// TwinCAT 3 PLC project PLC1
// ProgramVersion: 3.1.4026.19
// libraries:
//   Tc2_ControllerToolbox, * (Beckhoff Automation GmbH)
//   Tc2_PfwLib_Processing, * (Beckhoff Automation GmbH)
//   Tc2_Standard, * (Beckhoff Automation GmbH)
//   Tc2_System, * (Beckhoff Automation GmbH)
//   Tc2_Utilities, * (Beckhoff Automation GmbH)
//   Tc3_Module, * (Beckhoff Automation GmbH)
//   VisuDialogs, * (System)
// project tree:
//   / MAIN.TcPOU, MAIN_Fast.TcPOU, Visualization Manager.TcVMO (not stored)
//   Tasks/ Fast_Task.TcTTO, PLC_Task.TcTTO (not stored), Temperature_Task.TcTTO (not stored)
//   Temperature/DUTs/ E_HMIstatus.TcDUT, E_MainStateMachine.TcDUT, ST_TempLoad.TcDUT, ST_TempLoad_Cmd.TcDUT, ST_TempLoad_State.TcDUT, ST_TempSave.TcDUT, ST_TempSave_Cmd.TcDUT (not stored)
//   Temperature/ FB_Load.TcPOU, FB_MainVisu.TcPOU, FB_Save.TcPOU, TemperatureCtrl.TcPOU
//   Temperature/GVLs/ GVL_10_Visu.TcGVL (not stored), GVL_20_Application.TcGVL, GVL_30_Scope.TcGVL (not stored)
//   Temperature/TextLists/ GlobalTextList_1.TcGTLO (not stored), TL_Mparams_LREAL.TcTLO, TL_Params_BOOL.TcTLO (not stored), TL_Params_Enum.TcTLO (not stored), TL_Params_INT.TcTLO, TL_Pparmas.TcTLO (not stored), TL_Supply.TcTLO, TL_TcPfw_ErrorId.TcTLO, TL_TctrlOutSelect.TcTLO (not stored), TL_TctrlPowerTerminal.TcTLO (not stored), TL_TempSensType.TcTLO, TL_TerminalType.TcTLO (not stored)
//   Temperature/VISUs/DUTs/ st_ParamsUnsave.TcDUT (not stored), ST_Param_Visu.TcDUT (not stored)
//   Temperature/VISUs/POUs/ FB_Visu_Param.TcPOU (not stored), FB_Visu_Pparam.TcPOU (not stored), FB_Visu_Supply.TcPOU (not stored)
//   Temperature/VISUs/VISUs/Pages/Load Save/ Visu_SaveLoad.TcVIS
//   Temperature/VISUs/VISUs/Pages/LoopTest/ Visu_LoopTest.TcVIS
//   Temperature/VISUs/VISUs/Pages/Machine/Parameter/ Param_BOOL.TcVIS, Param_DINT.TcVIS, Param_ENUM_PowerTerm.TcVIS, Param_ENUM_SelOut.TcVIS, Param_ENUM_SensType.TcVIS, Param_ENUM_TermType.TcVIS, Param_LREAL.TcVIS
//   Temperature/VISUs/VISUs/Pages/Machine/Subpage/ Visu_Mparam_Autotune.TcVIS, Visu_Mparam_Cool.TcVIS, Visu_Mparam_Extruder.TcVIS (excluded from build), Visu_Mparam_General.TcVIS, Visu_Mparam_Heat.TcVIS, Visu_Mparam_Supply.TcVIS, Visu_Mparam_Temperature.TcVIS
//   Temperature/VISUs/VISUs/Pages/Machine/ Visu_MParam.TcVIS
//   Temperature/VISUs/VISUs/Pages/Product/ Param_LREAL_Pparam.TcVIS, Visu_PParam.TcVIS, Visu_PParam_Params.TcVIS
//   Temperature/VISUs/VISUs/Pages/Supply/ Param_LREAL_Supply.TcVIS, Visu_Supply.TcVIS, Visu_Supply_Params.TcVIS
//   Temperature/VISUs/VISUs/Pages/ Visu_Main.TcVIS
//   Utility/Linearisation/ FB_Linear_Interpolation.TcPOU
//   Utility/Ramp Generator/ FB_Ramp_Generator.TcPOU, ST_Ramp_Generator.TcDUT
//   Utility/Setpoint Generator/ FB_Setpoint_Generator.TcPOU, ST_Setpoint_Generator.TcDUT
// real-time tasks:
//   TASK Temperature Task: cycle T#25000us, priority 20, ADS port 350
//   TASK PLC Task: cycle T#10ms, priority 1, ADS port 351
//   TASK Fast Task: cycle T#2ms, priority 2, ADS port 352
// I/O:
//   DEVICE Device 1 (EtherCAT) (disabled), AmsNetId 5.70.226.154.2.1
//     Term 1 (EK1200) [EK1200-5000 EtherCAT Power supply (2A E-Bus)]
//       Term 2 (EL3202) [EL3202 2Ch. Ana. Input PT100 (RTD)]
//       Term 3 (EL1809) [EL1809 16Ch. Dig. Input 24V, 3ms]
//       Term 4 (EL2809) [EL2809 16Ch. Dig. Output 24V, 0.5A]
//       Term 5 (EL9011) [EL9011 End Terminal]
//   DEVICE Device 2 (EtherCAT Automation Protocol) (disabled), AmsNetId 5.77.2.52.3.1
//     Box 6 (Publisher)
//     Box 7 (Subscriber)

CONFIGURATION PLC1
    RESOURCE PLC ON TwinCAT3
        TASK Fast_Task(INTERVAL := T#2ms, PRIORITY := 2);
        PROGRAM MAIN_Fast WITH Fast_Task : MAIN_Fast;
    END_RESOURCE
END_CONFIGURATION

// ---- Temperature/DUTs/E_HMIstatus.TcDUT
TYPE E_HMIstatus :
(
	Off 				:= 0,
	Standby,
	On,
	Autotune,
	IdleLoad
);
END_TYPE

// ---- Temperature/DUTs/E_MainStateMachine.TcDUT
TYPE E_MainStateMachine :
(
	eMainSM_BasicInit 						:= 0,
	eMainSM_TempInit,
	eMainSM_MParamLoad,
	eMainSM_PParamLoad,
	eMainSM_SupParamLoad,
	eMainSM_StartUp,
	eMainSM_Idle
);
END_TYPE

// ---- Temperature/DUTs/ST_TempLoad.TcDUT
TYPE ST_TempLoad :
STRUCT
	stTempCmd						: ST_TempLoad_Cmd;
	stTempState						: ST_TempLoad_State;
END_STRUCT
END_TYPE

// ---- Temperature/DUTs/ST_TempLoad_Cmd.TcDUT
TYPE ST_TempLoad_Cmd :
STRUCT
	bLoadPparams							: BOOL;
	bLoadMparams							: BOOL;
	bLoadSupplyParams						: BOOL;
END_STRUCT
END_TYPE

// ---- Temperature/DUTs/ST_TempLoad_State.TcDUT
TYPE ST_TempLoad_State :
STRUCT
	bPparamLoaded									: BOOL;
	bMparamLoaded									: BOOL;
	bPparamLoad										: BOOL;
	bMparamLoad										: BOOL;
	bSupplyParamsLoad								: BOOL;
	bSupplyParamsLoaded								: BOOL;
END_STRUCT
END_TYPE

// ---- Temperature/DUTs/ST_TempSave.TcDUT
TYPE ST_TempSave :
STRUCT
	stTempCmd							: ST_TempSave_Cmd;
END_STRUCT
END_TYPE

// ---- Utility/Ramp Generator/ST_Ramp_Generator.TcDUT
TYPE ST_Ramp_Generator :
STRUCT
	tRefreshRate									: LREAL;
	fVelPos											: LREAL	:= 20;
	fVelNeg											: LREAL	:= 40;
END_STRUCT
END_TYPE

// ---- Utility/Setpoint Generator/ST_Setpoint_Generator.TcDUT
TYPE ST_Setpoint_Generator :
STRUCT
	tRefreshRate									: LREAL;
	bDisableRamping									: BOOL	:= FALSE;(*A continuous output value is not calculated if this parameter is TRUE. There is a step change between the output values*)
END_STRUCT
END_TYPE

// ---- Temperature/GVLs/GVL_20_Application.TcGVL
VAR_GLOBAL
	stTempLoad				: ST_TempLoad;
	stTempSave				: ST_TempSave;
END_VAR

// ---- MAIN_Fast.TcPOU
PROGRAM MAIN_Fast
VAR
	fbGetCurTaskIdx 			: GETCURTASKINDEX;
	bFirstCycle					: BOOL;
//	For temperature feedback linearisation
	fbLinInterpolation			: FB_Linear_Interpolation;
//	Setpoint generator
	fbSetpointGenerator			: FB_Setpoint_Generator;
//	Ramp generator
	fbRampGenerator				: FB_Ramp_Generator;
END_VAR


// =========================================================
	// Get plc task first cycle flag	
fbGetCurTaskIdx(); 
bFirstCycle:= _TaskInfo[fbGetCurTaskIdx.index].FirstCycle;

IF bFirstCycle THEN
	;
END_IF

	// Temperature feedback linearisation	
fbLinInterpolation();	
fbLinInterpolation.M_Cyclic();

	// Setpoint generator	
fbSetpointGenerator();
fbSetpointGenerator.M_Cyclic();	
	// Ramp generator
fbRampGenerator();
fbRampGenerator.M_Cyclic();
	
// =========================================================

END_PROGRAM

// ---- Utility/Linearisation/FB_Linear_Interpolation.TcPOU
FUNCTION_BLOCK FB_Linear_Interpolation
VAR CONSTANT
	nNoOfRows											: INT:= 45;
	nNoOfColumns										: INT:= 2;
END_VAR
VAR
	arrTableOffset										: ARRAY[1..nNoOfRows,1..nNoOfColumns] OF LREAL;	
	arrTable											: ARRAY[1..nNoOfRows,1..nNoOfColumns] OF LREAL;
	fIn, fOut, fManValue								: LREAL;
	bExtrapolate										: BOOL;
	eMode												: E_CTRL_MODE;
	stCTRL_LIN_INTERPOLATION_PARAMS						: ST_CTRL_LIN_INTERPOLATION_PARAMS;
	eErrorId											: E_CTRL_ERRORCODES;
	bError												: BOOL;
	fbCTRL_LIN_INTERPOLATION							: FB_CTRL_LIN_INTERPOLATION;
	bInit, bUpdate										: BOOL	:= TRUE;
	fbGetCurTaskIdx 									: GETCURTASKINDEX;
	bFirstCycle											: BOOL;
	fCycleTime											: LREAL := 0.025;
END_VAR

// =========================================================
	// Get temperature task first cycle flag	
fbGetCurTaskIdx(); 
bFirstCycle:= _TaskInfo[fbGetCurTaskIdx.index].FirstCycle;

IF bFirstCycle THEN
	;
END_IF

// Get Cycle Time
IF(GETCURTASKINDEXEX()<=0)THEN
	fCycletime:= TO_LREAL(0.025);(* Don't know, just guessing *)
ELSE
	fCycletime:= UDINT_TO_LREAL(_TaskInfo[GETCURTASKINDEXEX()].cycleTime)/10000000.0;
END_IF

// =========================================================

//FB_Init is always available implicitly and it is used primarily for initialization.
//The return value is not evaluated. For a specific influence, you can also declare the
//methods explicitly and provide additional code there with the standard initialization
//code. You can evaluate the return value.
METHOD FB_Init: BOOL
VAR_INPUT
    bInitRetains: BOOL; // TRUE: the retain variables are initialized (reset warm / reset cold)
    bInCopyCode: BOOL;  // TRUE: the instance will be copied to the copy code afterward (online change)   
END_VAR
// =========================================================
	// Init
	arrTableOffset[1,1]:= 0.1;		arrTableOffset[1,2]:= 0.9;
	arrTableOffset[2,1]:= 0.3;		arrTableOffset[2,2]:= 0.8;
	arrTableOffset[3,1]:= 0.5;		arrTableOffset[3,2]:= 0.7;
	arrTableOffset[4,1]:= 0.7;		arrTableOffset[4,2]:= 0.6;
	arrTableOffset[5,1]:= 0.9;		arrTableOffset[5,2]:= 0.5;
	arrTableOffset[6,1]:= 0.8;		arrTableOffset[6,2]:= 0.4;
	arrTableOffset[7,1]:= 0.7;		arrTableOffset[7,2]:= 0.3;
	arrTableOffset[8,1]:= 0.6;		arrTableOffset[8,2]:= 0.2;
	arrTableOffset[9,1]:= 0.5;		arrTableOffset[9,2]:= 0.1;
	arrTableOffset[10,1]:= 0.4;		arrTableOffset[10,2]:= 0.3;
	arrTableOffset[11,1]:= 0.3;		arrTableOffset[11,2]:= 0.5;
	arrTableOffset[12,1]:= 0.2;		arrTableOffset[12,2]:= 0.7;
	arrTableOffset[13,1]:= 0.1;		arrTableOffset[13,2]:= 0.9;
	arrTableOffset[14,1]:= 0.3;		arrTableOffset[14,2]:= 0.7;
	arrTableOffset[15,1]:= 0.5;		arrTableOffset[15,2]:= 0.5;
	arrTableOffset[16,1]:= 0.7;		arrTableOffset[16,2]:= 0.3;
	arrTableOffset[17,1]:= 0.9;		arrTableOffset[17,2]:= 0.1;
	arrTableOffset[18,1]:= 0.8;		arrTableOffset[18,2]:= 0.2;
	arrTableOffset[19,1]:= 0.7;		arrTableOffset[19,2]:= 0.3;
	arrTableOffset[20,1]:= 0.6;		arrTableOffset[20,2]:= 0.4;
	arrTableOffset[21,1]:= 0.5;		arrTableOffset[21,2]:= 0.5;
	arrTableOffset[22,1]:= 0.4;		arrTableOffset[22,2]:= 0.6;
	arrTableOffset[23,1]:= 0.3;		arrTableOffset[23,2]:= 0.7;
	arrTableOffset[24,1]:= 0.2;		arrTableOffset[24,2]:= 0.8;
	arrTableOffset[25,1]:= 0.1;		arrTableOffset[25,2]:= 0.9;
	arrTableOffset[26,1]:= 0.9;		arrTableOffset[26,2]:= 0.7;
	arrTableOffset[27,1]:= 0.7;		arrTableOffset[27,2]:= 0.5;
	arrTableOffset[28,1]:= 0.5;		arrTableOffset[28,2]:= 0.5;
	arrTableOffset[29,1]:= 0.3;		arrTableOffset[29,2]:= 0.3;
	arrTableOffset[30,1]:= 0.1;		arrTableOffset[30,2]:= 0.1;
	arrTableOffset[31,1]:= 0.3;		arrTableOffset[31,2]:= 0.3;
	arrTableOffset[32,1]:= 0.5;		arrTableOffset[32,2]:= 0.5;
	arrTableOffset[33,1]:= 0.7;		arrTableOffset[33,2]:= 0.7;
	arrTableOffset[34,1]:= 0.9;		arrTableOffset[34,2]:= 0.9;
	arrTableOffset[35,1]:= 0.8;		arrTableOffset[35,2]:= 0.7;
	arrTableOffset[36,1]:= 0.7;		arrTableOffset[36,2]:= 0.5;
	arrTableOffset[37,1]:= 0.6;		arrTableOffset[37,2]:= 0.3;
	arrTableOffset[38,1]:= 0.5;		arrTableOffset[38,2]:= 0.1;
	arrTableOffset[39,1]:= 0.4;		arrTableOffset[39,2]:= 0.2;
	arrTableOffset[40,1]:= 0.3;		arrTableOffset[40,2]:= 0.3;
	arrTableOffset[41,1]:= 0.2;		arrTableOffset[41,2]:= 0.4;
	arrTableOffset[42,1]:= 0.1;		arrTableOffset[42,2]:= 0.5;
	arrTableOffset[43,1]:= 0.3;		arrTableOffset[43,2]:= 0.6;
	arrTableOffset[44,1]:= 0.5;		arrTableOffset[44,2]:= 0.7;
	arrTableOffset[45,1]:= 0.7;		arrTableOffset[45,2]:= 0.8;
	
// =========================================================
END_METHOD

METHOD PUBLIC M_Cyclic
VAR_INPUT
END_VAR
// =========================================================
bUpdate := TRUE;

IF bInit OR bUpdate THEN
	(* Init array with the interpolation points  *)
	(* 	fIn					 						|		fOut		*)
	arrTable[1,1] := 25.0+arrTableOffset[1,1];			arrTable[1,2] := 25.0+arrTableOffset[1,2];
	arrTable[2,1] := 30.0+arrTableOffset[2,1];			arrTable[2,2] := 30.0+arrTableOffset[2,2];
	arrTable[3,1] := 35.0+arrTableOffset[3,1];			arrTable[3,2] := 35.0+arrTableOffset[3,2];
	arrTable[4,1] := 40.0+arrTableOffset[4,1];			arrTable[4,2] := 40.0+arrTableOffset[4,2];
	arrTable[5,1] := 45.0+arrTableOffset[5,1];			arrTable[5,2] := 45.0+arrTableOffset[5,2];
	arrTable[6,1] := 50.0+arrTableOffset[6,1];			arrTable[6,2] := 50.0+arrTableOffset[6,2];
	arrTable[7,1] := 55.0+arrTableOffset[7,1];			arrTable[7,2] := 55.0+arrTableOffset[7,2];
	arrTable[8,1] := 60.0+arrTableOffset[8,1];			arrTable[8,2] := 60.0+arrTableOffset[8,2];
	arrTable[9,1] := 65.0+arrTableOffset[9,1];			arrTable[9,2] := 65.0+arrTableOffset[9,2];
	arrTable[10,1] := 70.0+arrTableOffset[10,1];		arrTable[10,2] := 70.0+arrTableOffset[10,2];
	arrTable[11,1] := 75.0+arrTableOffset[11,1];		arrTable[11,2] := 75.0+arrTableOffset[11,2];
	arrTable[12,1] := 80.0+arrTableOffset[12,1];		arrTable[12,2] := 80.0+arrTableOffset[12,2];
	arrTable[13,1] := 85.0+arrTableOffset[13,1];		arrTable[13,2] := 85.0+arrTableOffset[13,2];
	arrTable[14,1] := 90.0+arrTableOffset[14,1];		arrTable[14,2] := 90.0+arrTableOffset[14,2];
	arrTable[15,1] := 95.0+arrTableOffset[15,1];		arrTable[15,2] := 95.0+arrTableOffset[15,2];
	arrTable[16,1] := 100.0+arrTableOffset[16,1];		arrTable[16,2] := 100.0+arrTableOffset[16,2];
	arrTable[17,1] := 105.0+arrTableOffset[17,1];		arrTable[17,2] := 105.0+arrTableOffset[17,2];
	arrTable[18,1] := 110.0+arrTableOffset[18,1];		arrTable[18,2] := 110.0+arrTableOffset[18,2];
	arrTable[19,1] := 115.0+arrTableOffset[19,1];		arrTable[19,2] := 115.0+arrTableOffset[19,2];
	arrTable[20,1] := 120.0+arrTableOffset[20,1];		arrTable[20,2] := 120.0+arrTableOffset[20,2];
	arrTable[21,1] := 125.0+arrTableOffset[21,1];		arrTable[21,2] := 125.0+arrTableOffset[21,2];
	arrTable[22,1] := 130.0+arrTableOffset[22,1];		arrTable[22,2] := 130.0+arrTableOffset[22,2];
	arrTable[23,1] := 135.0+arrTableOffset[23,1];		arrTable[23,2] := 135.0+arrTableOffset[23,2];
	arrTable[24,1] := 140.0+arrTableOffset[24,1];		arrTable[24,2] := 140.0+arrTableOffset[24,2];
	arrTable[25,1] := 145.0+arrTableOffset[25,1];		arrTable[25,2] := 145.0+arrTableOffset[25,2];
	arrTable[26,1] := 150.0+arrTableOffset[26,1];		arrTable[26,2] := 150.0+arrTableOffset[26,2];
	arrTable[27,1] := 155.0+arrTableOffset[27,1];		arrTable[27,2] := 155.0+arrTableOffset[27,2];
	arrTable[28,1] := 160.0+arrTableOffset[28,1];		arrTable[28,2] := 160.0+arrTableOffset[28,2];
	arrTable[29,1] := 165.0+arrTableOffset[29,1];		arrTable[29,2] := 165.0+arrTableOffset[29,2];
	arrTable[30,1] := 170.0+arrTableOffset[30,1];		arrTable[30,2] := 170.0+arrTableOffset[30,2];
	arrTable[31,1] := 175.0+arrTableOffset[31,1];		arrTable[31,2] := 175.0+arrTableOffset[31,2];
	arrTable[32,1] := 180.0+arrTableOffset[32,1];		arrTable[32,2] := 180.0+arrTableOffset[32,2];
	arrTable[33,1] := 185.0+arrTableOffset[33,1];		arrTable[33,2] := 185.0+arrTableOffset[33,2];
	arrTable[34,1] := 190.0+arrTableOffset[34,1];		arrTable[34,2] := 190.0+arrTableOffset[34,2];
	arrTable[35,1] := 195.0+arrTableOffset[35,1];		arrTable[35,2] := 195.0+arrTableOffset[35,2];
	arrTable[36,1] := 200.0+arrTableOffset[36,1];		arrTable[36,2] := 200.0+arrTableOffset[36,2];
	arrTable[37,1] := 205.0+arrTableOffset[37,1];		arrTable[37,2] := 205.0+arrTableOffset[37,2];
	arrTable[38,1] := 210.0+arrTableOffset[38,1];		arrTable[38,2] := 210.0+arrTableOffset[38,2];
	arrTable[39,1] := 215.0+arrTableOffset[39,1];		arrTable[39,2] := 215.0+arrTableOffset[39,2];
	arrTable[40,1] := 220.0+arrTableOffset[40,1];		arrTable[40,2] := 220.0+arrTableOffset[40,2];
	arrTable[41,1] := 225.0+arrTableOffset[41,1];		arrTable[41,2] := 225.0+arrTableOffset[41,2];
	arrTable[42,1] := 230.0+arrTableOffset[42,1];		arrTable[42,2] := 230.0+arrTableOffset[42,2];
	arrTable[43,1] := 235.0+arrTableOffset[43,1];		arrTable[43,2] := 235.0+arrTableOffset[43,2];
	arrTable[44,1] := 240.0+arrTableOffset[44,1];		arrTable[44,2] := 240.0+arrTableOffset[44,2];
	arrTable[45,1] := 245.0+arrTableOffset[45,1];		arrTable[45,2] := 245.0+arrTableOffset[45,2];;

	(* Init parameter struct *)
	stCTRL_LIN_INTERPOLATION_PARAMS.tCtrlCycleTime	:= UDINT_TO_TIME(_TaskInfo[GETCURTASKINDEXEX()].cycleTime/10000);
	stCTRL_LIN_INTERPOLATION_PARAMS.tTaskCycleTime	:= UDINT_TO_TIME(_TaskInfo[GETCURTASKINDEXEX()].cycleTime/10000);
	stCTRL_LIN_INTERPOLATION_PARAMS.nDataTable_NumberOfRows	:= nNoOfRows;

	(* Set the mode to ACTIVE --> Normal operation *)
	eMode := E_CTRL_MODE.eCTRL_MODE_ACTIVE;

	(* Reset the init flag *)
	bInit := FALSE;
	(* Reset the update flag *)
	bUpdate := FALSE;
END_IF

(* Set the address *)
stCTRL_LIN_INTERPOLATION_PARAMS.pDataTable_ADR			:= ADR(arrTable);
stCTRL_LIN_INTERPOLATION_PARAMS.nDataTable_SIZEOF		:= SIZEOF(arrTable);

(* Call interpolation fb *)
fbCTRL_LIN_INTERPOLATION(	fIn						:= fIn,
							fManValue				:= fManValue,
							bExtrapolate			:= bExtrapolate,
							stParams				:= stCTRL_LIN_INTERPOLATION_PARAMS,
							eMode					:= eMode,
							fOut					=> fOut,
							eErrorId				=> eErrorId,
							bError					=> bError);
							
// =========================================================
END_METHOD

END_FUNCTION_BLOCK

// ---- Utility/Setpoint Generator/FB_Setpoint_Generator.TcPOU
FUNCTION_BLOCK FB_Setpoint_Generator
VAR CONSTANT
	nNoOfRows											: INT:= 45;
END_VAR
VAR
	fManValue											: LREAL;
	eMode												: E_CTRL_MODE;
	nSetpointIndex										: INT:= 3;
	fCurrentSetpoint									: LREAL;
	bValueReached										: BOOL;

	fbCTRL_SETPOINT_GENERATOR							: FB_CTRL_SETPOINT_GENERATOR;
	stCTRL_SETPOINT_GENERATOR_PARAMS					: ST_CTRL_SETPOINT_GENERATOR_PARAMS;
	arrSetpointTable									: ARRAY [1..nNoOfRows] OF FLOAT;

	eErrorId											: E_CTRL_ERRORCODES;
	bError												: BOOL;

	bInit, bUpdate										: BOOL	:= TRUE;
	fbTON												: TON;
	
	fbGetCurTaskIdx 									: GETCURTASKINDEX;
	bFirstCycle											: BOOL;
	fCycleTime											: LREAL := 0.025;
	StSetPointGeneraor									: ST_Setpoint_Generator;
//	Scope
	fInToScope											: LREAL;
	fOutToScope											: LREAL;
END_VAR

// =========================================================
	// Get task first cycle flag	
fbGetCurTaskIdx(); 
bFirstCycle:= _TaskInfo[fbGetCurTaskIdx.index].FirstCycle;

IF bFirstCycle THEN
	;
END_IF

// Get Cycle Time
IF(GETCURTASKINDEXEX()<=0)THEN
	fCycletime:= TO_LREAL(0.025);(* Don't know, just guessing *)
ELSE
	fCycletime:= UDINT_TO_LREAL(_TaskInfo[GETCURTASKINDEXEX()].cycleTime)/10000000.0;
END_IF

// =========================================================

//FB_Init is always available implicitly and it is used primarily for initialization.
//The return value is not evaluated. For a specific influence, you can also declare the
//methods explicitly and provide additional code there with the standard initialization
//code. You can evaluate the return value.
METHOD FB_Init: BOOL
VAR_INPUT
    bInitRetains: BOOL; // TRUE: the retain variables are initialized (reset warm / reset cold)
    bInCopyCode: BOOL;  // TRUE: the instance will be copied to the copy code afterward (online change)   
END_VAR
// =========================================================
(* Init the setpoint array *)
arrSetpointTable[ 1 ]	:= 25;
arrSetpointTable[ 2 ]	:= 30;
arrSetpointTable[ 3 ]	:= 35;
arrSetpointTable[ 4 ]	:= 40;
arrSetpointTable[ 5 ]	:= 45;
arrSetpointTable[ 6 ]	:= 50;
arrSetpointTable[ 7 ]	:= 55;
arrSetpointTable[ 8 ]	:= 60;
arrSetpointTable[ 9 ]	:= 65;
arrSetpointTable[ 10 ]	:= 70;
arrSetpointTable[ 11 ]	:= 75;
arrSetpointTable[ 12 ]	:= 80;
arrSetpointTable[ 13 ]	:= 85;
arrSetpointTable[ 14 ]	:= 90;
arrSetpointTable[ 15 ]	:= 95;
arrSetpointTable[ 16 ]	:= 100;
arrSetpointTable[ 17 ]	:= 105;
arrSetpointTable[ 18 ]	:= 110;
arrSetpointTable[ 19 ]	:= 115;
arrSetpointTable[ 20 ]	:= 120;
arrSetpointTable[ 21 ]	:= 125;
arrSetpointTable[ 22 ]	:= 130;
arrSetpointTable[ 23 ]	:= 135;
arrSetpointTable[ 24 ]	:= 140;
arrSetpointTable[ 25 ]	:= 145;
arrSetpointTable[ 26 ]	:= 150;
arrSetpointTable[ 27 ]	:= 155;
arrSetpointTable[ 28 ]	:= 160;
arrSetpointTable[ 29 ]	:= 165;
arrSetpointTable[ 30 ]	:= 170;
arrSetpointTable[ 31 ]	:= 175;
arrSetpointTable[ 32 ]	:= 180;
arrSetpointTable[ 33 ]	:= 185;
arrSetpointTable[ 34 ]	:= 190;
arrSetpointTable[ 35 ]	:= 195;
arrSetpointTable[ 36 ]	:= 200;
arrSetpointTable[ 37 ]	:= 205;
arrSetpointTable[ 38 ]	:= 210;
arrSetpointTable[ 39 ]	:= 215;
arrSetpointTable[ 40 ]	:= 220;
arrSetpointTable[ 41 ]	:= 225;
arrSetpointTable[ 42 ]	:= 230;
arrSetpointTable[ 43 ]	:= 235;
arrSetpointTable[ 44 ]	:= 240;
arrSetpointTable[ 45 ]	:= 245;

(*
(* Init parameter struct *)
stCTRL_SETPOINT_GENERATOR_PARAMS.tTaskCycleTime				:= UDINT_TO_TIME(_TaskInfo[GETCURTASKINDEXEX()].cycleTime/10000);
stCTRL_SETPOINT_GENERATOR_PARAMS.tCtrlCycleTime				:= UDINT_TO_TIME(_TaskInfo[GETCURTASKINDEXEX()].cycleTime/10000);
stCTRL_SETPOINT_GENERATOR_PARAMS.bDisableRamping			:= FALSE;
stCTRL_SETPOINT_GENERATOR_PARAMS.fVeloNeg					:= 10;
stCTRL_SETPOINT_GENERATOR_PARAMS.fVeloPos					:= 8;
stCTRL_SETPOINT_GENERATOR_PARAMS.nDataTable_NumberOfRows	:= 4;

(* Set the mode to ACTIVE --> normal operation *)
eMode := eCTRL_MODE_ACTIVE;
*)
// =========================================================
END_METHOD

METHOD PUBLIC M_Cyclic
VAR_INPUT
END_VAR
// =========================================================
IF bInit OR bUpdate THEN
	(* Init parameter struct *)
	stCTRL_SETPOINT_GENERATOR_PARAMS.tTaskCycleTime				:= UDINT_TO_TIME(_TaskInfo[GETCURTASKINDEXEX()].cycleTime/10000);
	stCTRL_SETPOINT_GENERATOR_PARAMS.tCtrlCycleTime				:= UDINT_TO_TIME(_TaskInfo[GETCURTASKINDEXEX()].cycleTime/10000);
	stCTRL_SETPOINT_GENERATOR_PARAMS.bDisableRamping			:= FALSE; 
	stCTRL_SETPOINT_GENERATOR_PARAMS.fVeloNeg					:= 10; (* In units per second *)
	stCTRL_SETPOINT_GENERATOR_PARAMS.fVeloPos					:= 8;  (* In units per second *)
	stCTRL_SETPOINT_GENERATOR_PARAMS.nDataTable_NumberOfRows	:= nNoOfRows;

	(* Set the mode to ACTIVE --> normal operation *)
	eMode := eCTRL_MODE_ACTIVE;
	(* Reset the init flag *)
	bInit := FALSE;
	(* Reset the update flag *)
	bUpdate := FALSE;
END_IF

(* Set the address *)
stCTRL_SETPOINT_GENERATOR_PARAMS.nDataTable_SIZEOF			:= SIZEOF(arrSetpointTable);
stCTRL_SETPOINT_GENERATOR_PARAMS.pDataTable_ADR				:= ADR(arrSetpointTable);

(* Generate setpoint-index *)
fbTON( IN := TRUE, PT:= T#5S);
IF fbTON.Q
THEN
	nSetpointIndex	:=  nSetpointIndex + 1;
	IF nSetPointIndex > nNoOfRows
	THEN
		nSetPointIndex := 1;
	END_IF
	fbTON( IN := FALSE);
END_IF

(* Copy var to scope var *)
fInToScope := INT_TO_FLOAT(nSetpointIndex);

(* Call setpointgenerator *)
fbCTRL_SETPOINT_GENERATOR(nSetpointIndex:= nSetpointIndex,
										fManValue				:= fManValue,
										eMode					:= eMode,
										stParams				:= stCTRL_SETPOINT_GENERATOR_PARAMS,
										fOut					=> fCurrentSetpoint,
										bValueReached		=> bValueReached
										 );

(* Copy var to scope var *)
fOutToScope := fCurrentSetpoint;

// =========================================================
END_METHOD

END_FUNCTION_BLOCK

// ---- Utility/Ramp Generator/FB_Ramp_Generator.TcPOU
FUNCTION_BLOCK FB_Ramp_Generator
VAR CONSTANT
END_VAR
VAR
	(* Input *)
	bEnable												: BOOL		:= TRUE;
	fStart												: LREAL;
	fTarget												: LREAL		:= 	50.0;
	(* Output *)
	fOut												: LREAL;
	bValueReached										: BOOL;
	(* Function block *)
	fbCTRL_RAMP_GENERATOR								: FB_CTRL_RAMP_GENERATOR;
	stCTRL_RAMP_GENERATOR_PARAMS						: ST_CTRL_RAMP_GENERATOR_PARAMS;
	eErrorId											: E_CTRL_ERRORCODES;
	bError												: BOOL;
	bInit, bUpdate										: BOOL	:= TRUE;
	fbTON												: TON;	
	fbGetCurTaskIdx 									: GETCURTASKINDEX;
	bFirstCycle											: BOOL;
	fCycleTime											: LREAL := 0.025;
	stRampGenerator										: ST_Ramp_Generator;
//	Scope
	fInToScope											: LREAL;
	fOutToScope											: LREAL;
END_VAR

// =========================================================
	// Get task first cycle flag	
fbGetCurTaskIdx(); 
bFirstCycle:= _TaskInfo[fbGetCurTaskIdx.index].FirstCycle;

IF bFirstCycle THEN
	;
END_IF

// Get Cycle Time
IF(GETCURTASKINDEXEX()<=0)THEN
	fCycletime:= TO_LREAL(0.025);(* Don't know, just guessing *)
ELSE
	fCycletime:= UDINT_TO_LREAL(_TaskInfo[GETCURTASKINDEXEX()].cycleTime)/10000000.0;
END_IF

// =========================================================

//FB_Init is always available implicitly and it is used primarily for initialization.
//The return value is not evaluated. For a specific influence, you can also declare the
//methods explicitly and provide additional code there with the standard initialization
//code. You can evaluate the return value.
METHOD FB_Init: BOOL
VAR_INPUT
    bInitRetains: BOOL; // TRUE: the retain variables are initialized (reset warm / reset cold)
    bInCopyCode: BOOL;  // TRUE: the instance will be copied to the copy code afterward (online change)   
END_VAR
// =========================================================
	(* Init parameter struct *)
	stCTRL_RAMP_GENERATOR_PARAMS.tTaskCycleTime		:= T#10MS;
	stCTRL_RAMP_GENERATOR_PARAMS.tCtrlCycleTime		:= T#10MS;
	stCTRL_RAMP_GENERATOR_PARAMS.fVeloPos			:= 20; (* in units per second *)
	stCTRL_RAMP_GENERATOR_PARAMS.fVeloNeg			:= 40; (* in units per second *)

// =========================================================
END_METHOD

METHOD PUBLIC M_Cyclic
VAR_INPUT
END_VAR
// =========================================================
IF bInit OR bUpdate THEN
	(* Init parameter struct *)
	stCTRL_RAMP_GENERATOR_PARAMS.tTaskCycleTime		:= UDINT_TO_TIME(_TaskInfo[GETCURTASKINDEXEX()].cycleTime/10000);
	stCTRL_RAMP_GENERATOR_PARAMS.tCtrlCycleTime		:= UDINT_TO_TIME(_TaskInfo[GETCURTASKINDEXEX()].cycleTime/10000);
	stCTRL_RAMP_GENERATOR_PARAMS.fVeloPos			:= 20; (* In units per second *)
	stCTRL_RAMP_GENERATOR_PARAMS.fVeloNeg			:= 40; (* In units per second *)
	(* Reset the init flag *)
	bInit := FALSE;
	(* Reset the update flag *)
	bUpdate := FALSE;
END_IF

(* Generate target value *)
fbTON(IN:= TRUE, PT	:= T#6S);	
IF fbTON.Q THEN
	fTarget := -1.0 * fTarget;
	fbTON(	 IN	:= FALSE);
END_IF

(* Copy var to scope var *)
fInToScope := fTarget;

(* Call function block *)
fbCTRL_RAMP_GENERATOR(	bEnable			:= bEnable,
						fStart			:= fStart,
						fTarget			:= fTarget,
						stParams		:= stCTRL_RAMP_GENERATOR_PARAMS,
						fOut			=> fOut,
						bValueReached	=> bValueReached,
						bError			=> bError,
						eErrorId		=> eErrorId);

(* Copy var to scope var *)
fOutToScope := fOut;

// =========================================================
END_METHOD

END_FUNCTION_BLOCK

// ---- MAIN.TcPOU
{attribute 'TcCallAfterOutputUpdate'}
PROGRAM MAIN
VAR
	fbGetCurTaskIdx 			: GETCURTASKINDEX;
	bFirstCycle					: BOOL;
	lrAbsHigh	: lreal;
END_VAR

// =========================================================
	// Get plc task first cycle flag	
fbGetCurTaskIdx(); 
bFirstCycle:= _TaskInfo[fbGetCurTaskIdx.index].FirstCycle;

IF bFirstCycle THEN
	;
END_IF

// =========================================================

END_PROGRAM

// ---- Temperature/FB_Load.TcPOU
FUNCTION_BLOCK FB_Load
VAR
	nCount							: INT;
END_VAR

// =========================================================
(* Product parameters *)
(* Product parameter - Set load on true *)
IF (stTempLoad.stTempCmd.bLoadPparams AND NOT stTempLoad.stTempState.bPparamLoad) THEN
	stTempLoad.stTempCmd.bLoadPparams:=
	stTempLoad.stTempState.bPparamLoaded:= FALSE;
	stTempLoad.stTempState.bPparamLoad:= TRUE;
	FOR nCount:=cnPfwTempCtrlFirst TO cnPfwTempCtrlLast DO
		aaaPfwTempPparamFromHmi[nCount].bLoadParams:= TRUE;
	END_FOR
END_IF
(* Product parameter - check load is done *)
IF stTempLoad.stTempState.bPparamLoad THEN
	stTempLoad.stTempState.bPparamLoad:= FALSE;
	FOR nCount:=cnPfwTempCtrlFirst TO cnPfwTempCtrlLast DO
		IF aaaPfwTempPparamFromHmi[nCount].bLoadParams THEN
			stTempLoad.stTempState.bPparamLoad:= TRUE;
		END_IF
	END_FOR
	stTempLoad.stTempState.bPparamLoaded:= NOT stTempLoad.stTempState.bPparamLoad;
END_IF

(* Machine parameters *)
(* Machine parameter - Set load on true *)
IF (stTempLoad.stTempCmd.bLoadMparams AND NOT stTempLoad.stTempState.bMparamLoad) THEN
	stTempLoad.stTempCmd.bLoadMparams:=
	stTempLoad.stTempState.bMparamLoaded:= FALSE;
	stTempLoad.stTempState.bMparamLoad:= TRUE;
	FOR nCount:=cnPfwTempCtrlFirst TO cnPfwTempCtrlLast DO
		aaaPfwTempMparamFromHmi[nCount].bLoadParams:= TRUE;
	END_FOR
END_IF
(* Machine parameter - check load is done *)
IF stTempLoad.stTempState.bMparamLoad THEN
	stTempLoad.stTempState.bMparamLoad:= FALSE;
	FOR nCount:=cnPfwTempCtrlFirst TO cnPfwTempCtrlLast DO
		IF aaaPfwTempMparamFromHmi[nCount].bLoadParams THEN
			stTempLoad.stTempState.bPparamLoad:= TRUE;
		END_IF
	END_FOR
	stTempLoad.stTempState.bMparamLoaded:= NOT stTempLoad.stTempState.bMparamLoad;
END_IF


(* Supply lines *)
(* Supply lines - Set load on true *)
IF (stTempLoad.stTempCmd.bLoadSupplyParams AND NOT stTempLoad.stTempState.bSupplyParamsLoad) THEN
	stTempLoad.stTempCmd.bLoadSupplyParams:=
	stTempLoad.stTempState.bSupplyParamsLoaded:= FALSE;
	stTempLoad.stTempState.bSupplyParamsLoad:= TRUE;
	FOR nCount:=cnPfwAppSupplyFirst TO cnPfwAppSupplyLast DO
		stPfwSupplyLineCfg[nCount].bLoadParams:= TRUE;
	END_FOR
END_IF
(* Supply lines - check load is done *)
IF stTempLoad.stTempState.bSupplyParamsLoad THEN
	stTempLoad.stTempState.bSupplyParamsLoad:= FALSE;
	FOR nCount:=cnPfwAppSupplyFirst TO cnPfwAppSupplyLast DO
		IF stPfwSupplyLineCfg[nCount].bLoadParams THEN
			stTempLoad.stTempState.bSupplyParamsLoad:= TRUE;
		END_IF
	END_FOR
	stTempLoad.stTempState.bSupplyParamsLoaded:= NOT stTempLoad.stTempState.bSupplyParamsLoad;
END_IF
// =========================================================

END_FUNCTION_BLOCK

// ---- Temperature/FB_MainVisu.TcPOU
FUNCTION_BLOCK FB_MainVisu
VAR
	bOldVisuNext									: BOOL;
	ncount											: INT;
	bAutotuneAllDone								: BOOL;
	eOldState										: E_HMIstatus;
	bEntry											: BOOL := TRUE;
	nIdx											: INT;
	fbVisuMParam									: FB_Visu_Param;
	fbVisuPParam									: FB_Visu_PParam;
	fbVisuSupply									: FB_Visu_Supply;
END_VAR

// =========================================================
//
//		All Zones
//

bEntry:= (eStatus<>eOldState);
eOldState:= eStatus;

CASE eStatus OF

	Off:
		IF bEntry THEN
			FOR ncount:=cnPfwTempCtrlFirst TO cnPfwTempCtrlLast DO
				aaaPfwTempMparamFromHmi[ncount].Enable:= FALSE;
				stPfwTempCtrl[nCount].Enable:= FALSE;
			END_FOR
			bEntry:= FALSE;
		END_IF
	
	Standby:
		IF bEntry THEN
			FOR ncount:=cnPfwTempCtrlFirst TO cnPfwTempCtrlLast DO
				IF aaaPfwTempToHmi[nCount].InUse THEN
					stPfwTempCtrl[nCount].SelSetpoint:= TRUE;
					aaaPfwTempMparamFromHmi[ncount].Enable:= TRUE;
					stPfwTempCtrl[nCount].Enable:= TRUE;
				END_IF
			END_FOR
			bEntry:= FALSE;
		END_IF
	
	On:
		IF bEntry THEN
			FOR ncount:=cnPfwTempCtrlFirst TO cnPfwTempCtrlLast DO
				IF aaaPfwTempToHmi[nCount].InUse THEN
					stPfwTempCtrl[nCount].SelSetpoint:= FALSE;
					aaaPfwTempMparamFromHmi[ncount].Enable:= TRUE;
					stPfwTempCtrl[nCount].Enable:= TRUE;
				END_IF
			END_FOR
			bEntry:=FALSE;
		END_IF
	
	Autotune:
		IF bEntry THEN
			FOR ncount:=cnPfwTempCtrlFirst TO cnPfwTempCtrlLast DO
				IF aaaPfwTempToHmi[nCount].InUse THEN
					stPfwTempCtrl[nCount].Enable:= TRUE;
					aaaPfwTempMparamFromHmi[ncount].Enable:= TRUE;
					aaaPfwTempMparamFromHmi[ncount].Autotune:= TRUE;
				END_IF
			END_FOR
		ELSE
			bAutotuneAllDone:=TRUE;
			FOR ncount:=cnPfwTempCtrlFirst TO cnPfwTempCtrlLast DO
				IF(aaaPfwTempToHmi[nCount].TuningDone OR aaaPfwTempToHmi[nCount].Error) THEN
					IF aaaPfwTempToHmi[nCount].InUse THEN
						stPfwTempCtrl[nCount].Enable:= FALSE;
						aaaPfwTempMparamFromHmi[ncount].Enable:= FALSE;
						aaaPfwTempMparamFromHmi[ncount].Autotune:= FALSE;
					END_IF
				ELSE
					bAutoTuneAllDone:= FALSE;
				END_IF
			END_FOR
			IF bAutotuneAllDone THEN
				eStatus:= Standby;
			END_IF
		END_IF
		
	IdleLoad:
		IF bEntry THEN
			FOR ncount:=cnPfwTempCtrlFirst TO cnPfwTempCtrlLast DO
				IF aaaPfwTempToHmi[ncount].Enable THEN
					aaaPfwTempMparamFromHmi[ncount].Ena_TuneIdleLoad:= TRUE;
				END_IF
			END_FOR
		ELSE
			FOR ncount:=cnPfwTempCtrlFirst TO cnPfwTempCtrlLast DO
				bVisuIdleLoadAktiv:= FALSE;
				IF(aaaPfwTempToHmi[ncount].IdleLoadActive)THEN
					bVisuIdleLoadAktiv:= TRUE;
				END_IF
			END_FOR
			IF NOT bVisuIdleLoadAktiv THEN
				eStatus:= On;
			END_IF
		END_IF
END_CASE


//
//		Selected Zone
//

// Select Zone
IF(bVisuNext)THEN
	nVisuCount:= MIN(nVisuCount+1,cnPfwTempCtrlLast);
	bVisuNext:= FALSE;
ELSIF(bVisuBefore)THEN
	nVisuCount:= MAX(nVisuCount-1,cnPfwTempCtrlFirst);
	bVisuBefore:= FALSE;
END_IF

IF(bVisuAutotune)THEN
	aaaPfwTempMparamFromHmi[nVisuCount].Autotune:= TRUE;
ELSIF bVisuIdleLoad THEN
	aaaPfwTempMparamFromHmi[nVisuCount].Ena_TuneIdleLoad:= TRUE;
END_IF


ErrorHandling();
fbVisuMParam(stMParam_Visu:=stMParam_Visu, stParamsUnsave:=stParamsUnsave);
fbVisuPParam(stPParam_Visu:=stPParam_Visu, stParamsUnsave:=stParamsUnsave);
fbVisuSupply(stSupply_Visu:=stSupply_Visu, stParamsUnsave:=stParamsUnsave);

// =========================================================

ACTION ErrorHandling:
// =========================================================
bGlobalError:= FALSE;
sErrorText:= 'No Error';
FOR ncount:=cnPfwTempCtrlFirst TO cnPfwTempCtrlLast DO
	IF aaaPfwTempToHmi[ncount].Error THEN
		IF sErrorText= 'No Error' THEN
			sErrorText:= 'Error in Zone ';
		ELSE
			sErrorText:= CONCAT(sErrorText, ', ');
		END_IF
		sErrorText:= CONCAT(sErrorText, INT_TO_STRING(ncount));
		bGlobalError:= TRUE;
	END_IF
END_FOR
// =========================================================
END_ACTION

END_FUNCTION_BLOCK

// ---- Temperature/FB_Save.TcPOU
FUNCTION_BLOCK FB_Save
VAR
	nCount												: INT;
	bSavePparamsOld										: BOOL;
	bSaveMparamsOld										: BOOL;
	bSaveSupplyOld										: BOOL;
END_VAR

// =========================================================
(* Save product parameters *)
IF(stTempSave.stTempCmd.bSavePparams AND NOT bSavePparamsOld)  THEN
	FOR nCount:=cnPfwTempCtrlFirst TO cnPfwTempCtrlLast DO
		IF	aaaPfwTempPparamFromHmi[nCount].SaveDelay= -1 THEN
			aaaPfwTempPparamFromHmi[nCount].SaveDelay:= 100_000;
		END_IF
	END_FOR
ELSIF(stTempSave.stTempCmd.bSavePparams AND  bSavePparamsOld)  THEN
	stTempSave.stTempCmd.bSavePparams:= FALSE;
	FOR nCount:=cnPfwTempCtrlFirst TO cnPfwTempCtrlLast DO
		IF	aaaPfwTempPparamFromHmi[nCount].SaveDelay>-1 THEN
			stTempSave.stTempCmd.bSavePparams:= TRUE;
		END_IF
	END_FOR
END_IF
bSavePparamsOld:= stTempSave.stTempCmd.bSavePparams;


(* Save machine parameters *)
IF(stTempSave.stTempCmd.bSaveMparams AND NOT bSaveMparamsOld)  THEN
	FOR nCount:=cnPfwTempCtrlFirst TO cnPfwTempCtrlLast DO
		IF	aaaPfwTempMparamFromHmi[nCount].SaveDelay= -1 THEN
			aaaPfwTempMparamFromHmi[nCount].SaveDelay:= 100_000;
		END_IF
	END_FOR
ELSIF(stTempSave.stTempCmd.bSaveMparams AND bSaveMparamsOld)  THEN
	stTempSave.stTempCmd.bSaveMparams:= FALSE;
	FOR nCount:=cnPfwTempCtrlFirst TO cnPfwTempCtrlLast DO
		IF	aaaPfwTempMparamFromHmi[nCount].SaveDelay>-1 THEN
			stTempSave.stTempCmd.bSaveMparams:= TRUE;
		END_IF
	END_FOR
	IF NOT stTempSave.stTempCmd.bSaveMparams THEN
		;
	END_IF
END_IF
bSaveMparamsOld:= stTempSave.stTempCmd.bSaveMparams;


(* Save supply lines *)
IF(stTempSave.stTempCmd.bSaveSupplyParams AND NOT bSaveSupplyOld)  THEN
	FOR nCount:=cnPfwAppSupplyFirst TO cnPfwAppSupplyLast DO
		IF	stPfwSupplyLineCfg[nCount].SaveDelay= -1 THEN
			stPfwSupplyLineCfg[nCount].SaveDelay:= 100_000;
		END_IF
	END_FOR
ELSIF(stTempSave.stTempCmd.bSaveSupplyParams AND  bSaveSupplyOld)  THEN
	stTempSave.stTempCmd.bSaveSupplyParams:= FALSE;
	FOR nCount:=cnPfwAppSupplyFirst TO cnPfwAppSupplyLast DO
		IF	stPfwSupplyLineCfg[nCount].SaveDelay>-1 THEN
			stTempSave.stTempCmd.bSaveSupplyParams:= TRUE;
		END_IF
	END_FOR
END_IF
bSaveSupplyOld:= stTempSave.stTempCmd.bSaveSupplyParams;

// =========================================================

END_FUNCTION_BLOCK

// ---- Temperature/TemperatureCtrl.TcPOU
PROGRAM TemperatureCtrl
VAR
	eState						: E_MainStateMachine := eMainSM_BasicInit;
	nCount						: INT := 0;
	fCycleTime					: LREAL := 0.025;
	fbTempCtrl					: FB_TempCtrlMainBody_TcPfw_TC3;
	fbVisu						: FB_MainVisu;
	bEntry						: BOOL;
	fbSave						: FB_Save;
	fbLoad						: FB_Load;

	fbGetCurTaskIdx 			: GETCURTASKINDEX;
	bFirstCycle					: BOOL;
END_VAR

// =========================================================
	// Get temperature task first cycle flag	
fbGetCurTaskIdx(); 
bFirstCycle:= _TaskInfo[fbGetCurTaskIdx.index].FirstCycle;

IF bFirstCycle THEN
	;
END_IF

// =========================================================
	// Temp
///aaaPfwTempMparamFromHmi[1].SensorType:= eTcPfwTempSensT_TC_K;
///aaaPfwTempMparamFromHmi[1].TempSensTerm:= eTcPfwTermT_EL331x;
///	iRead						: INT;
///	opHeat 				AT %Q*	: BOOL;
/// opCool				AT %Q*	: BOOL:
///TcPfw_Global_TempCtrlVariables.in_PfwTempCtrlInput[1].EL_SnsData:= iRead;
///opHeat :=out_PfwTempCtrlOutput[1].SelOutPos;
///opCool :=out_PfwTempCtrlOutput[1].SelOutNeg;

// =========================================================
CASE eState OF	
	E_MainStateMachine.eMainSM_BasicInit:
		_01_BasicInit();
		bEntry:= TRUE;
		eState:= E_MainStateMachine.eMainSM_MParamLoad;
		
	E_MainStateMachine.eMainSM_TempInit:
		_02_ParamsInit();
		bParamsInit:= FALSE;
		eState:= E_MainStateMachine.eMainSM_Idle;
		
	E_MainStateMachine.eMainSM_MParamLoad:
		IF bEntry THEN
			bEntry:= FALSE;
			stTempLoad.stTempCmd.bLoadMparams:= TRUE;
		ELSE
			IF stTempLoad.stTempState.bMparamLoaded THEN
				eState:= E_MainStateMachine.eMainSM_PParamLoad;
				bEntry:= TRUE;
			END_IF
		END_IF
	
	E_MainStateMachine.eMainSM_PParamLoad:
		IF bEntry THEN
			bEntry:= FALSE;
			stTempLoad.stTempCmd.bLoadPparams:= TRUE;
		ELSE
			IF stTempLoad.stTempState.bPparamLoaded THEN
				eState:= E_MainStateMachine.eMainSM_SupParamLoad;
				bEntry:= TRUE;
			END_IF
		END_IF
		
	E_MainStateMachine.eMainSM_SupParamLoad:
		IF bEntry THEN
			bEntry:= FALSE;
			stTempLoad.stTempCmd.bLoadSupplyParams:= TRUE;
		ELSE
			IF stTempLoad.stTempState.bSupplyParamsLoaded THEN
				eState:= E_MainStateMachine.eMainSM_StartUp;
				bEntry:= TRUE;
			END_IF
		END_IF
		
	E_MainStateMachine.eMainSM_StartUp:
		bEntry:= FALSE;
		fbTempCtrl.ConfigEnable:= TRUE;
		fbTempCtrl.tCycle:= fCycleTime;
		fbTempCtrl.Looptest_Enable:= FALSE;
		fbTempCtrl.Callback_Enable:= TRUE;
		fbTempCtrl.Simu_Enable:= TRUE;
		eState:= E_MainStateMachine.eMainSM_Idle;
	
	E_MainStateMachine.eMainSM_Idle:
		IF bParamsInit THEN
			eState:= E_MainStateMachine.eMainSM_TempInit;
		END_IF
		
END_CASE

// =========================================================
fbTempCtrl(
	Looptest_Enable:= TRUE,
	Scope_TempCtrlVariables:= Scope_TempCtrlVariables);
	
fbVisu();

fbSave();
fbLoad();

// =========================================================

ACTION _01_BasicInit:
// =========================================================
// Get Cycle Time
IF(GETCURTASKINDEXEX()<=0)THEN
	fCycletime:= TO_LREAL(0.025);(* Don't know, just guessing *)
ELSE
	fCycletime:= UDINT_TO_LREAL(_TaskInfo[GETCURTASKINDEXEX()].cycleTime)/10000000.0;
END_IF

// Init Zone ID/Name
FOR nCount := cnPfwTempCtrlFirst TO cnPfwTempCtrlLast DO
	aaaPfwTempMparamFromHmi[nCount].ZoneId := nCount;(* Zone id	*)
	aaaPfwTempMparamFromHmi[nCount].ZoneName := CONCAT('Zone_', INT_TO_STRING(nCount));(* Zone name  *)
END_FOR

// =========================================================
END_ACTION

ACTION _02_ParamsInit:
// =========================================================
(* Initialize of the machine parameters*)
	FOR nCount := cnPfwTempCtrlFirst TO cnPfwTempCtrlLast DO
		aaaPfwTempMparamFromHmi[nCount].AbsoluteHigh:= 300;											(* Limiting value of absolute hight.	*)
		aaaPfwTempMparamFromHmi[nCount].AbsoluteLow:= 100;											(* Limiting value of absolute low.	*)
		aaaPfwTempMparamFromHmi[nCount].InUse:= TRUE;												(* Zone is in use	*)
		aaaPfwTempMparamFromHmi[nCount].Enable:= TRUE;
		aaaPfwTempMparamFromHmi[nCount].SensorType:= E_TcPfw_TempSensType.eTcPfwTempSensT_NoSensor;	(* Simulation	*)
		aaaPfwTempMparamFromHmi[nCount].ExtruderId:= 1;												(* Simulation	*)
		aaaPfwTempMparamFromHmi[nCount].TempSensTerm:= 0;											(* Simulation	*)
		aaaPfwTempMparamFromHmi[nCount].ZoneId:= nCount;											(* Zone id		*)
		aaaPfwTempMparamFromHmi[nCount].ZoneName:= CONCAT('Zone_', INT_TO_STRING(nCount));			(* Zone name	*)
		IF(aaaPfwTempMparamFromHmi[nCount].KpCool<0.1)THEN
			aaaPfwTempMparamFromHmi[nCount].KpCool:= 0.1;											(* Default Kp cooling	*)
		END_IF
		IF(aaaPfwTempMparamFromHmi[nCount].KpHeat<0.1)THEN
			aaaPfwTempMparamFromHmi[nCount].KpHeat:= 0.2;											(* Default Kp heating 	*)
		END_IF
(*		aaaPfwTempMparamFromHmi[nCount].SettlingTime:= 5.0;											(* Settling Time	*)*)
//		aaaPfwTempMparamFromHmi[nCount].SupplyLoad_Cooler:= 100; 									(* Coolingpower	*)
		aaaPfwTempMparamFromHmi[nCount].SupplyLoad_Heater:= 1200;	 								(* Heatingpower	*)
		aaaPfwTempMparamFromHmi[nCount].TuneEnd:= 80;												(* Tune End % of setpoint	*)
		aaaPfwTempMparamFromHmi[nCount].TuneKp:= 1.2;												(* Kp Tuning	*)
		aaaPfwTempMparamFromHmi[nCount].TuneTd:= 0.25;												(* Td Tuning	*)
		aaaPfwTempMparamFromHmi[nCount].TuneTn:= 2;													(* Tn Tuning	*)
		aaaPfwTempMparamFromHmi[nCount].TuneTv:= 0.5;												(* Tv Tuning	*)
		aaaPfwTempMparamFromHmi[nCount].TuneY:= 100;												(* Y Tuning		*)
		aaaPfwTempMparamFromHmi[nCount].Ramping_Rate:= 0.005;										(* Ramping rate	*)
		aaaPfwTempMparamFromHmi[nCount].Ramping_Tolerance:= 10;										(* Ramping tolerance*)
		aaaPfwTempMparamFromHmi[nCount].OutputSel_H:= E_TcPfw_TctrlOutSelect.eTcPfwTcOut_PWM;		(* Heating output signal	*)
		aaaPfwTempMparamFromHmi[nCount].OutputSel_C:= E_TcPfw_TctrlOutSelect.eTcPfwTcOut_NoSignal;	(* Cooling output signal	*)
		aaaPfwTempMparamFromHmi[nCount].UseCooling:= FALSE;											(* Cooling on	*)
		aaaPfwTempMparamFromHmi[nCount].TuneCooling:= FALSE;										(* Cooling on	*)
		aaaPfwTempMparamFromHmi[nCount].ExtruderCompEna:= FALSE;									(* Extruder comp	*)
		aaaPfwTempMparamFromHmi[nCount].fc_Enable:= FALSE;											(* Zwangskuelung	*)
		aaaPfwTempMparamFromHmi[nCount].fc_OffTime:= 600.0;											(* Zwangskuelung	*)
		aaaPfwTempMparamFromHmi[nCount].fc_OnTime:= 10.0;											(* Zwangskuelung	*)

(*		aaaPfwTempMparamFromHmi[nCount].SupplyLoad_Tolerance:= 20.0;								(* Supply Tolerance	*)*)

		aaaPfwTempMparamFromHmi[nCount].SupplyLoad_Tolerance:= 0.0;									(* Supply Tolerance	*)

		aaaPfwTempMparamFromHmi[nCount].SupplyId:= 1;
		aaaPfwTempMparamFromHmi[nCount].ModuleId:= 1;
	END_FOR
	(* Mapping of the zones to the module and supply lines	*)
		//

	(* Initialize of the product parameter*)
	FOR nCount := cnPfwTempCtrlFirst TO cnPfwTempCtrlLast DO
		aaaPfwTempPparamFromHmi[nCount].Setpoint:= 180;
		aaaPfwTempPparamFromHmi[nCount].StandbySetpoint:= 18;
		aaaPfwTempPparamFromHmi[nCount].Threshold_M:= -10;
		aaaPfwTempPparamFromHmi[nCount].Threshold_MM:= -15;
		aaaPfwTempPparamFromHmi[nCount].Threshold_P:= 10;
		aaaPfwTempPparamFromHmi[nCount].Threshold_PP:= 15;
		aaaPfwTempPparamFromHmi[nCount].Update:= TRUE;
	END_FOR

	(* Initialize of the supply lines*)
	FOR nCount := cnPfwAppSupplyFirst TO cnPfwAppSupplyLast DO
		stPfwSupplyLineCfg[nCount].fPwmCycleTime:= 1;
		stPfwSupplyLineCfg[nCount].fPwmMaxOnTime:= 1.0;
		stPfwSupplyLineCfg[nCount].fPwmMinOnTime:= 0.1;
		stPfwSupplyLineCfg[nCount].fPwmMaxRampLoad:= 1;
		stPfwSupplyLineCfg[nCount].nPwmFactorC:= 10;
	END_FOR
	
// =========================================================
END_ACTION

END_PROGRAM

// ---- Temperature/TextLists/TL_Mparams_LREAL.TcTLO
TEXTLIST TL_Mparams_LREAL
  1 = 'AbsoluteHigh'
  2 = 'AbsoluteLow'
  3 = 'ExtruderComp'
  4 = 'KpCool'
  5 = 'KpHeat'
  6 = 'TdCool'
  7 = 'TdHeat'
  8 = 'TnCool'
  9 = 'TnHeat'
  10 = 'TvCool'
  11 = 'TvHeat'
  12 = 'Overshoot'
  13 = 'Tracking_Rate'
  14 = 'Tracking_Td'
  15 = 'Ramping_Rate'
  16 = 'Ramping_RateC'
  17 = 'Ramping_Tolerance'
  18 = 'dTmax'
  19 = 'SensorOffset'
  20 = 'SettlingTime'
  21 = 'SupplyLoad_Cooler'
  22 = 'SupplyLoad_Heater'
  23 = 'SupplyLoad_Tolerance'
  24 = 'TuneEnd'
  25 = 'TuneKp'
  26 = 'TuneTd'
  27 = 'TuneTn'
  28 = 'TuneTv'
  29 = 'TuneTrackingTd'
  30 = 'TuneY'
  31 = 'L_LoadIdle'
  32 = 'Weighting_C'
  33 = 'ErrorHeatingFactor'
  34 = 'fPwmStdMaxOnTime'
  35 = '*** not Used ***'
  36 = 'fPwmMinOnTime'
  37 = 'fc_OnTime'
  38 = 'fc_OffTime'
  39 = 'ActTempGain'
  40 = 'ActTempOffset'
  41 = 'SaveDelay'
   = ''
END_TEXTLIST

// ---- Temperature/TextLists/TL_Params_INT.TcTLO
TEXTLIST TL_Params_INT
  1 = 'App_HmiType'
  2 = 'TermChannel'
  3 = 'ExtruderId'
  4 = 'ModuleId'
  5 = 'ZoneId'
  6 = 'SupplyId'
  7 = 'CJ_CompMode'
  8 = 'CJ_CompZone'
  9 = 'SensTermSwapIdx'
  10 = 'HeaterSwapIdx'
  11 = 'CoolerSwapIdx'
  12 = 'nPwmFactorC'
  13 = '*** not Used ***'
  14 = '*** not Used ***'
  15 = '*** not Used ***'
  16 = '*** not Used ***'
  17 = '*** not Used ***'
  18 = '*** not Used ***'
  19 = '*** not Used ***'
  20 = '*** not Used ***'
  21 = '*** not Used ***'
  22 = '*** not Used ***'
  23 = '*** not Used ***'
  24 = '*** not Used ***'
  25 = '*** not Used ***'
  26 = '*** not Used ***'
  27 = '*** not Used ***'
  28 = '*** not Used ***'
  29 = '*** not Used ***'
  30 = '*** not Used ***'
  31 = '*** not Used ***'
  32 = '*** not Used ***'
  33 = '*** not Used ***'
  34 = '*** not Used ***'
  35 = '*** not Used ***'
  36 = '*** not Used ***'
  37 = '*** not Used ***'
  38 = '*** not Used ***'
  39 = '*** not Used ***'
  40 = '*** not Used ***'
   = ''
END_TEXTLIST

// ---- Temperature/TextLists/TL_Supply.TcTLO
TEXTLIST TL_Supply
  1 = 'fPwmCycleTime'
  2 = 'fPwmMinOnTime'
  3 = 'fPwmMaxOnTime'
  4 = 'fPwmMaxOnC'
  5 = 'fPwmMaxRampLoad'
  6 = 'fActSupplyLoad'
  7 = 'fActSupplyLoad'
  8 = 'fActSupplyCurrent'
  9 = 'fSupplyLoad'
  10 = 'fSupplyMatch'
   = ''
END_TEXTLIST

// ---- Temperature/TextLists/TL_TcPfw_ErrorId.TcTLO
TEXTLIST TL_TcPfw_ErrorId
  0 = 'dwTcPfwTempErrNoError'
  4098 = 'dwTcPfwTempErrBusy'
  4099 = 'dwTcPfwTempTuneErr_NoTravel'
  4100 = 'dwTcPfwTempTuneErr_NoSettling'
  4101 = 'dwTcPfwTempTuneErr_Aborted'
  4102 = 'dwTcPfwTempTuneErr_ShortOfPoints'
  4103 = 'dwTcPfwTempTuneErr_NoTop'
  4104 = ''
  4105 = 'dwTcPfwTempTuneErr_NoResponse'
  17508 = 'dwTcPfwTempErrSnsHdwFailed'
  20464 = 'dwTcPfwTempErrDisconected'
  20465 = 'dwTcPfwTempErr_NoResponse'
  20466 = 'dwTcPfwTempErrNotOperational\n'
  20467 = 'dwTcPfwTempErrIoSwapCollision\n'
  20468 = 'dwTcPfwTempErrAdsSwapCollision\n'
  20469 = 'dwTcPfwTempErrInheritedFault\n'
  20478 = 'dwTcPfwTempErrOverCurrent\n'
  20479 = 'dwTcPfwTempErrUnderCurrent'
  20480 = 'dwTcPfwTempErrSnsCommFailed'
  1800 = 'dwTcPfwTempErrBusy'
  17489 = 'dwTcPfwTempErrSnsOverrun\n'
   = ''
END_TEXTLIST

// ---- Temperature/TextLists/TL_TempSensType.TcTLO
TEXTLIST TL_TempSensType
  0 = 'NoSensor'
  1 = 'TC_B'
  2 = 'TC_E'
  3 = 'TC_J'
  4 = 'TC_K'
  5 = 'TC_L'
  6 = 'TC_N'
  7 = 'TC_R'
  8 = 'TC_S'
  9 = 'TC_T'
  10 = 'TC_U'
  100 = 'PT_100'
  101 = 'NI_100'
  102 = 'NI_120'
  103 = 'PT_200'
  104 = 'PT_500'
  105 = 'PT_1000'
  106 = 'NI_1000'
  10000 = 'Customized'
   = ''
END_TEXTLIST

// ---- Temperature/VISUs/VISUs/Pages/Load Save/Visu_SaveLoad.TcVIS
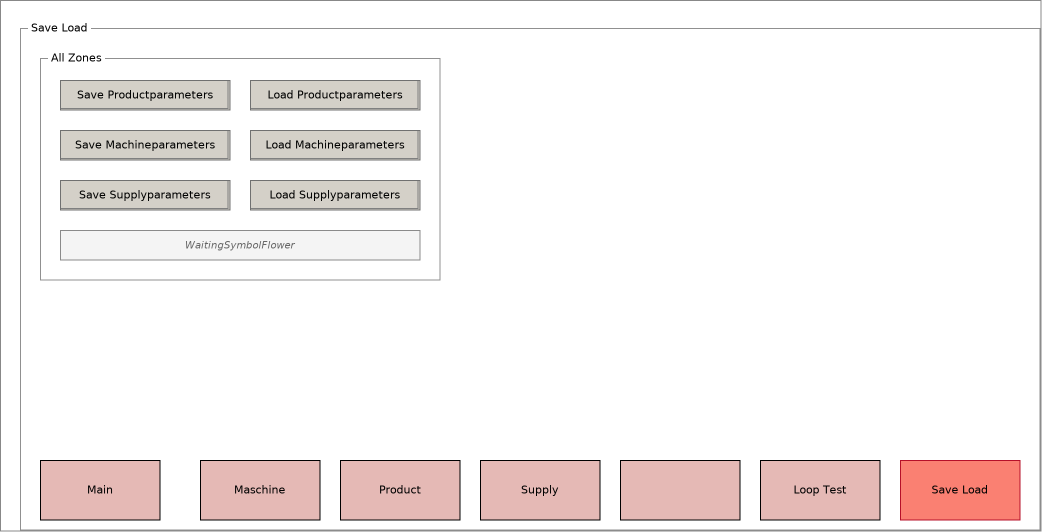
VISUALIZATION Visu_SaveLoad  // 1042x532
    GroupBox (20,20 1020x510), "Save Load"
        Rectangle (20,440 120x60), "Main"
            OnMouseClick: change screen: Visu_Main
        GroupBox (20,30 400x230), "All Zones", input disabled if: stTempSave.stTempCmd.bSaveMparams OR stTempSave.stTempCmd.bSaveSupplyParams OR stTempSave.stTempCmd.bSavePparams OR stTempLoad.stTempCmd.bLoadMparams OR stTempLoad.stTempCmd.bLoadPparams OR stTempLoad.stTempCmd.bLoadSupplyParams
            Button (20,30 170x30), "Save Productparameters"
                toggle stTempSave.stTempCmd.bSavePparams
            Button (210,30 170x30), "Load Productparameters"
                toggle stTempLoad.stTempCmd.bLoadPparams
            Button (20,80 170x30), "Save Machineparameters"
                toggle stTempSave.stTempCmd.bSaveMparams
            Button (210,80 170x30), "Load Machineparameters"
                toggle stTempLoad.stTempCmd.bLoadMparams
            Button (20,130 170x30), "Save Supplyparameters"
                toggle stTempSave.stTempCmd.bSaveSupplyParams
            Button (210,130 170x30), "Load Supplyparameters"
                toggle stTempLoad.stTempCmd.bLoadSupplyParams
            WaitingSymbolFlower (20,180 360x30), invisible if: NOT(stTempSave.stTempCmd.bSaveMparams OR stTempSave.stTempCmd.bSaveSupplyParams OR stTempSave.stTempCmd.bSavePparams OR stTempLoad.stTempCmd.bLoadMparams OR stTempLoad.stTempCmd.bLoadPparams OR stTempLoad.stTempCmd.bLoadSupplyParams)
        Rectangle (880,440 120x60), "Save Load"
            OnMouseClick: change screen: Visu_SaveLoad
        Rectangle (320,440 120x60), "Product"
            OnMouseClick: change screen: Visu_PParam
        Rectangle (180,440 120x60), "Maschine"
            OnMouseClick: change screen: Visu_MParam
        Rectangle (460,440 120x60), "Supply"
            OnMouseClick: change screen: Visu_Supply
        Rectangle (600,440 120x60)
        Rectangle (740,440 120x60), "Loop Test"
            OnMouseClick: change screen: Visu_LoopTest
END_VISUALIZATION

// ---- Temperature/VISUs/VISUs/Pages/LoopTest/Visu_LoopTest.TcVIS
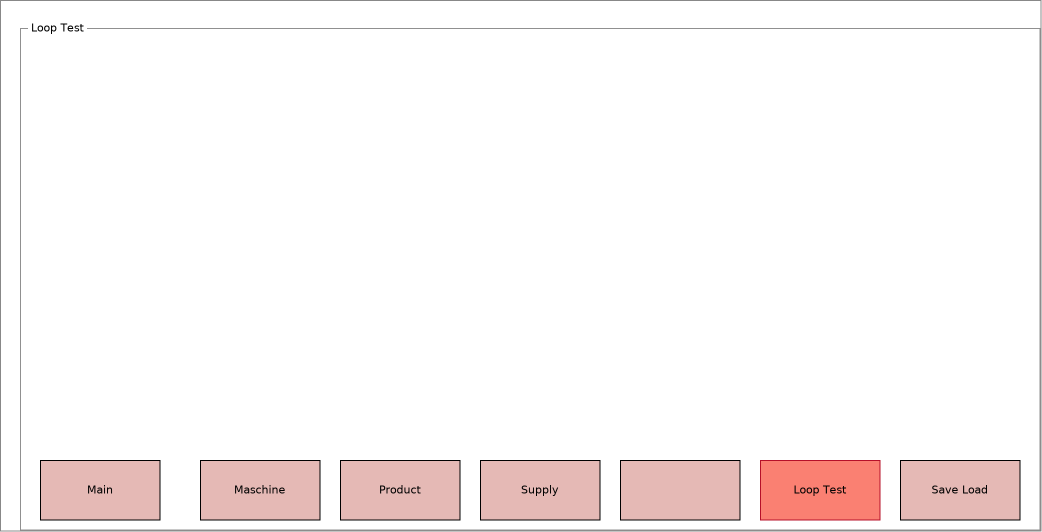
VISUALIZATION Visu_LoopTest  // 1042x532
    GroupBox (20,20 1020x510), "Loop Test"
        Rectangle (20,440 120x60), "Main"
            OnMouseClick: change screen: Visu_Main
        Rectangle (880,440 120x60), "Save Load"
            OnMouseClick: change screen: Visu_SaveLoad
        Rectangle (320,440 120x60), "Product"
            OnMouseClick: change screen: Visu_PParam
        Rectangle (180,440 120x60), "Maschine"
            OnMouseClick: change screen: Visu_MParam
        Rectangle (460,440 120x60), "Supply"
            OnMouseClick: change screen: Visu_Supply
        Rectangle (600,440 120x60)
        Rectangle (740,440 120x60), "Loop Test"
            OnMouseClick: change screen: Visu_LoopTest
END_VISUALIZATION

// ---- Temperature/VISUs/VISUs/Pages/Machine/Parameter/Param_BOOL.TcVIS
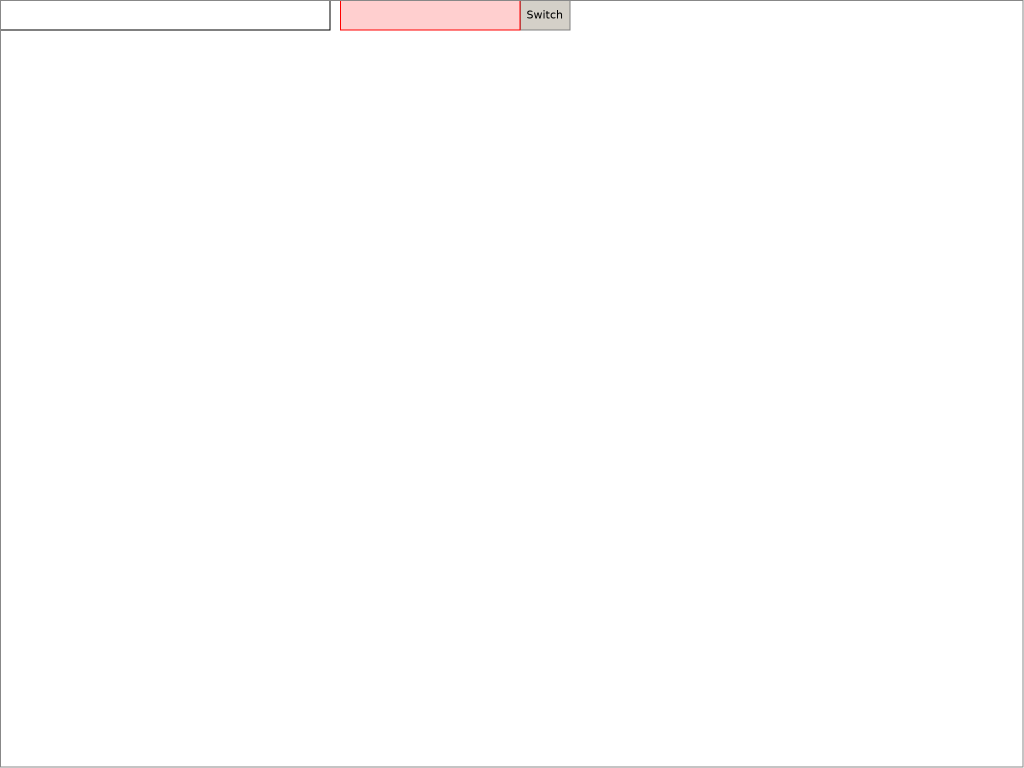
VISUALIZATION Param_BOOL  // 1024x768
    Rectangle (0,0 330x30), text list: 'TL_Params_BOOL', text index: nIdx
    Rectangle (520,0 50x30), "Switch", colour toggle: stMParam_Visu.bBoolSetValue[nIdx]
        OnMouseClick: execute { stMParam_Visu.bBoolSetValue[nIdx]:=TRUE; }
    Rectangle (340,0 180x30), colour toggle: stMParam_Visu.bBoolAktValue[nIdx]
    Rectangle (600,0 150x30)
END_VISUALIZATION

// ---- Temperature/VISUs/VISUs/Pages/Machine/Parameter/Param_DINT.TcVIS
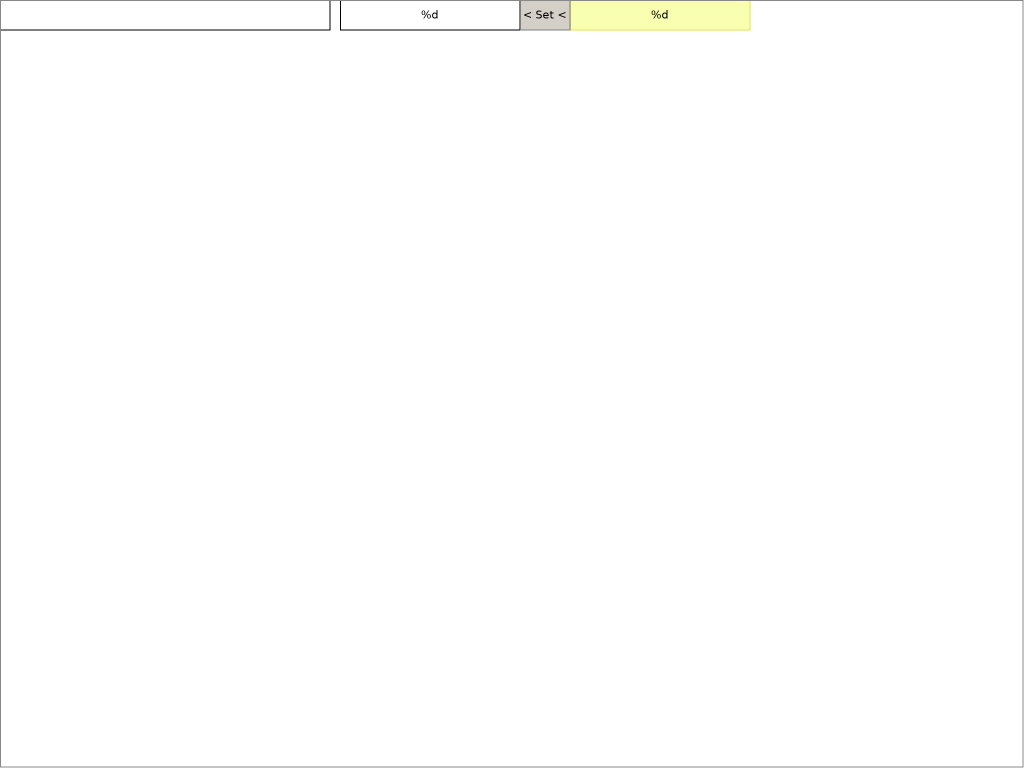
VISUALIZATION Param_DINT  // 1024x768
    Rectangle (340,0 180x30), "%d", text variable: stMParam_Visu.nDintAktValue[nIdx]
    Rectangle (0,0 330x30), text list: 'TL_Params_INT', text index: nIdx
    Rectangle (570,0 180x30), "%d", text variable: stMParam_Visu.nDintNewValue[nIdx]
        OnMouseClick: write the text variable via Default
    Rectangle (520,0 50x30), "< Set <"
        OnMouseClick: execute { stMParam_Visu.bDintSetValue[nIdx]:=TRUE; }
END_VISUALIZATION

// ---- Temperature/VISUs/VISUs/Pages/Machine/Parameter/Param_ENUM_PowerTerm.TcVIS
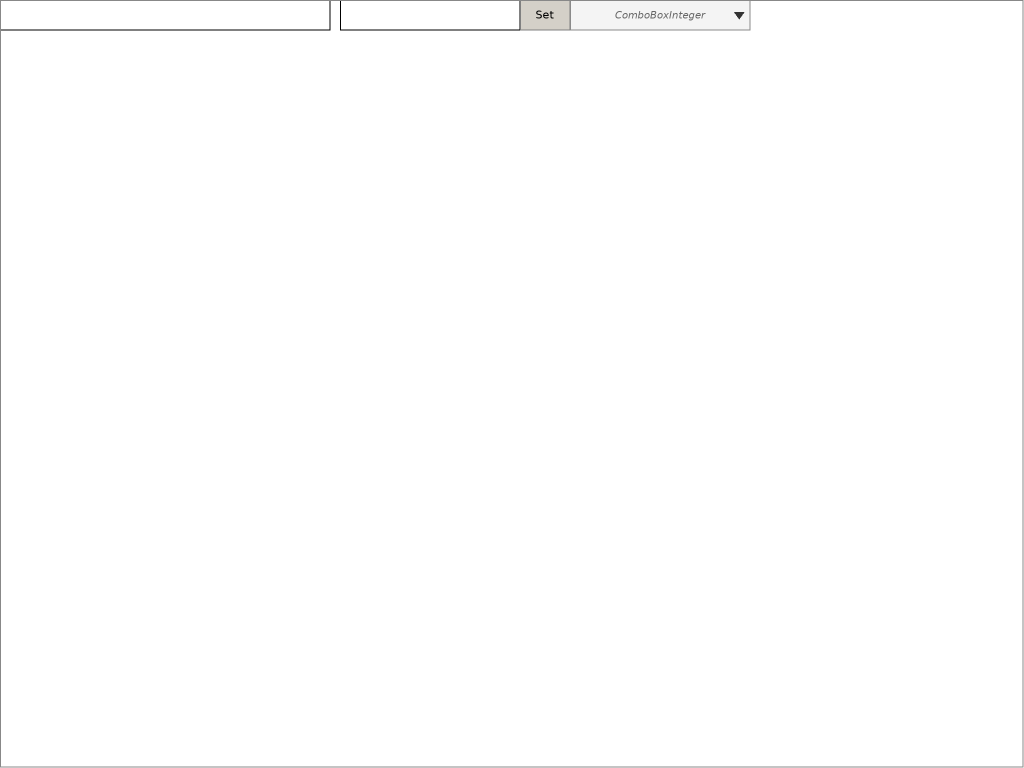
VISUALIZATION Param_ENUM_PowerTerm  // 1024x768
    Rectangle (340,0 180x30), text list: 'TL_TctrlPowerTerminal', text index: stMParam_Visu.nEnumAktValue[nIdx]
    Rectangle (0,0 330x30), text list: 'TL_Params_Enum', text index: nIdx
    Rectangle (520,0 50x30), "Set"
        OnMouseClick: execute { stMParam_Visu.bEnumSetValue[nIdx]:=TRUE; }
    ComboBoxInteger (570,0 180x30), variable: stMParam_Visu.nEnumNewValue[nIdx], text list: 'TL_TctrlPowerTerminal'
END_VISUALIZATION

// ---- Temperature/VISUs/VISUs/Pages/Machine/Parameter/Param_ENUM_SelOut.TcVIS
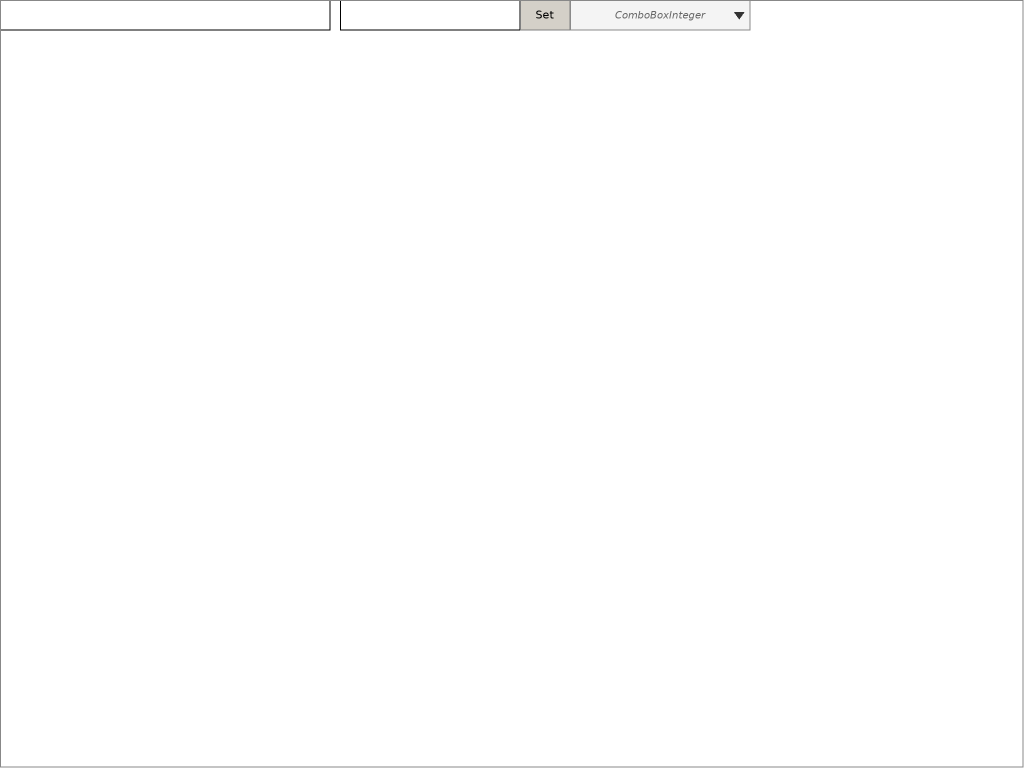
VISUALIZATION Param_ENUM_SelOut  // 1024x768
    Rectangle (340,0 180x30), text list: 'TL_TctrlOutSelect', text index: stMParam_Visu.nEnumAktValue[nIdx]
    Rectangle (0,0 330x30), text list: 'TL_Params_Enum', text index: nIdx
    Rectangle (520,0 50x30), "Set"
        OnMouseClick: execute { stMParam_Visu.bEnumSetValue[nIdx]:=TRUE; }
    ComboBoxInteger (570,0 180x30), variable: stMParam_Visu.nEnumNewValue[nIdx], text list: 'TL_TctrlOutSelect'
END_VISUALIZATION

// ---- Temperature/VISUs/VISUs/Pages/Machine/Parameter/Param_ENUM_SensType.TcVIS
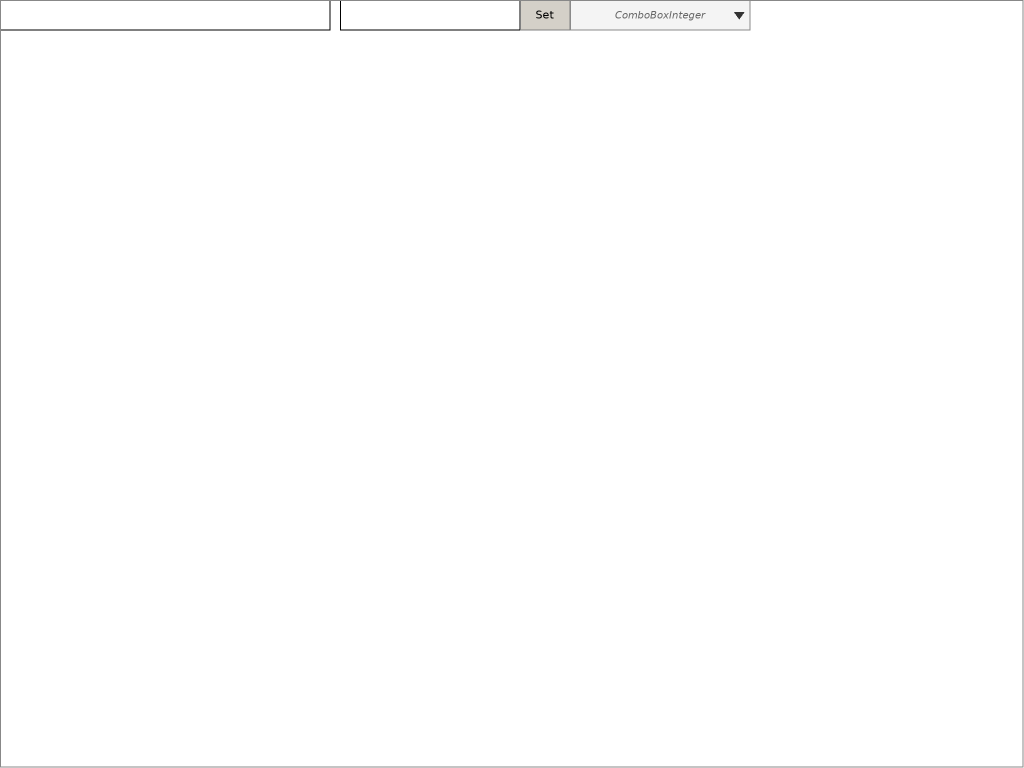
VISUALIZATION Param_ENUM_SensType  // 1024x768
    Rectangle (340,0 180x30), text list: 'TL_TempSensType', text index: stMParam_Visu.nEnumAktValue[nIdx]
    Rectangle (0,0 330x30), text list: 'TL_Params_Enum', text index: nIdx
    Rectangle (520,0 50x30), "Set"
        OnMouseClick: execute { stMParam_Visu.bEnumSetValue[nIdx]:=TRUE; }
    ComboBoxInteger (570,0 180x30), variable: stMParam_Visu.nEnumNewValue[nIdx], text list: 'TL_TempSensType'
END_VISUALIZATION

// ---- Temperature/VISUs/VISUs/Pages/Machine/Parameter/Param_ENUM_TermType.TcVIS
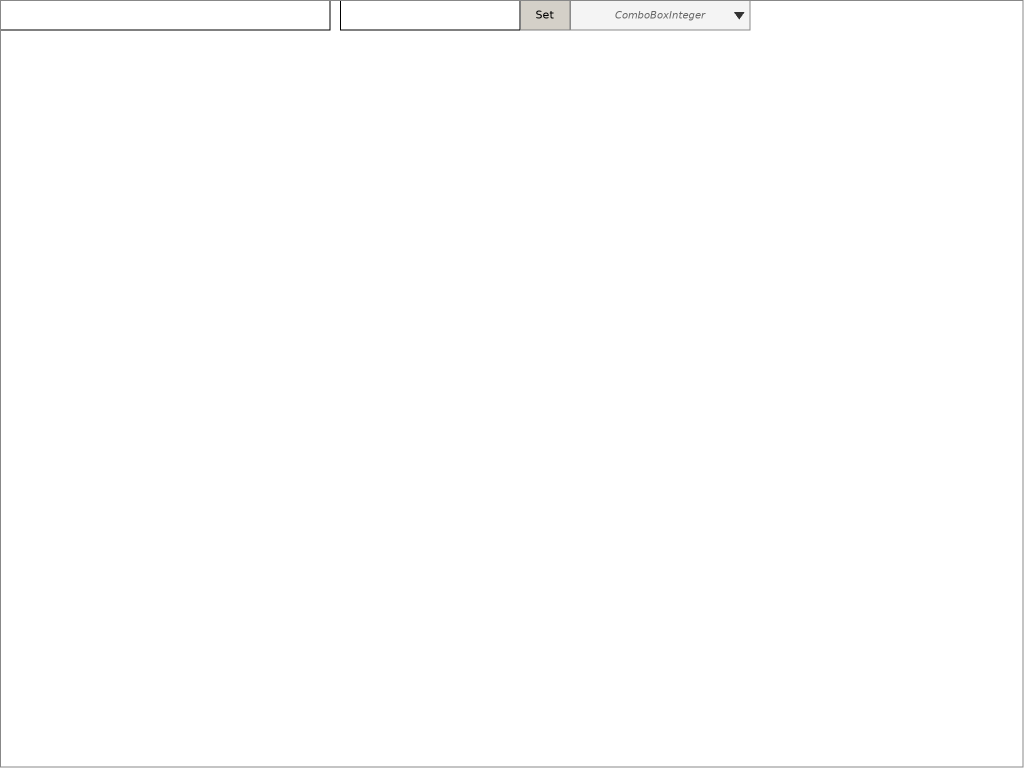
VISUALIZATION Param_ENUM_TermType  // 1024x768
    Rectangle (340,0 180x30), text list: 'TL_TerminalType', text index: stMParam_Visu.nEnumAktValue[nIdx]
    Rectangle (0,0 330x30), text list: 'TL_Params_Enum', text index: nIdx
    Rectangle (520,0 50x30), "Set"
        OnMouseClick: execute { stMParam_Visu.bEnumSetValue[nIdx]:=TRUE; }
    ComboBoxInteger (570,0 180x30), variable: stMParam_Visu.nEnumNewValue[nIdx], text list: 'TL_TerminalType'
END_VISUALIZATION

// ---- Temperature/VISUs/VISUs/Pages/Machine/Parameter/Param_LREAL.TcVIS
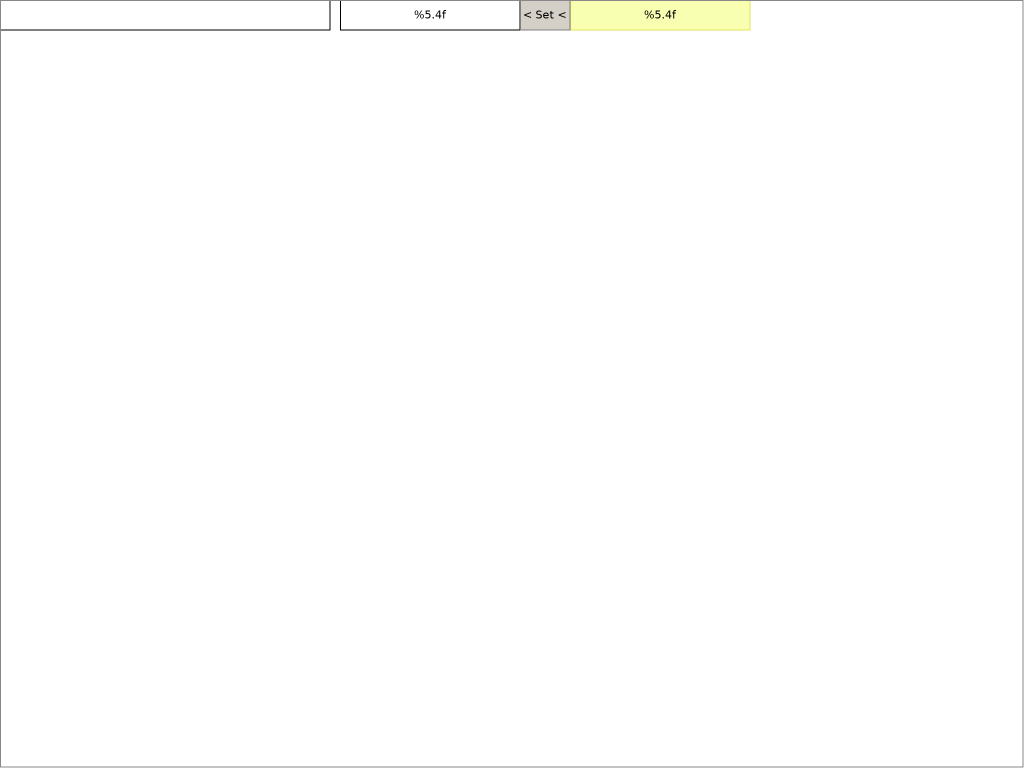
VISUALIZATION Param_LREAL  // 1024x768
    Rectangle (340,0 180x30), "%5.4f", text variable: stMParam_Visu.fLrealAktValue[nIdx]
    Rectangle (0,0 330x30), text list: 'TL_Mparams_LREAL', text index: nIdx
    Rectangle (570,0 180x30), "%5.4f", text variable: stMParam_Visu.fLrealNewValue[nIdx]
        OnMouseClick: write the text variable via Default
    Rectangle (520,0 50x30), "< Set <"
        OnMouseClick: execute { stMParam_Visu.bLrealSetValue[nIdx]:=TRUE; }
END_VISUALIZATION

// ---- Temperature/VISUs/VISUs/Pages/Machine/Subpage/Visu_Mparam_Autotune.TcVIS
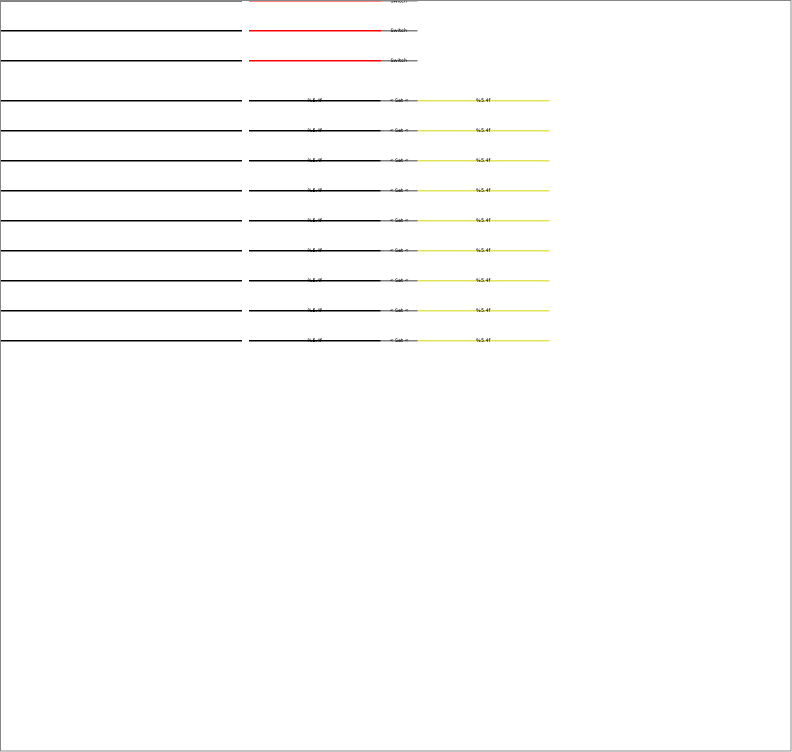
VISUALIZATION Visu_Mparam_Autotune  // 792x752
    Frame (0,100 750x30)
        shows Param_LREAL(nIdx := 24)
    Frame (0,130 750x30)
        shows Param_LREAL(nIdx := 25)
    Frame (0,160 750x30)
        shows Param_LREAL(nIdx := 26)
    Frame (0,190 750x30)
        shows Param_LREAL(nIdx := 27)
    Frame (0,220 750x30)
        shows Param_LREAL(nIdx := 28)
    Frame (0,250 750x30)
        shows Param_LREAL(nIdx := 29)
    Frame (0,280 750x30)
        shows Param_LREAL(nIdx := 30)
    Frame (0,310 750x30)
        shows Param_LREAL(nIdx := 31)
    Frame (0,340 750x30)
        shows Param_LREAL(nIdx := 23)
    Frame (0,60 750x30)
        shows Param_BOOL(nIdx := 10)
    Frame (0,30 750x30)
        shows Param_BOOL(nIdx := 4)
    Frame (0,0 750x30)
        shows Param_BOOL(nIdx := 5)
    Rectangle (40,720 750x30)
END_VISUALIZATION

// ---- Temperature/VISUs/VISUs/Pages/Machine/Subpage/Visu_Mparam_Cool.TcVIS
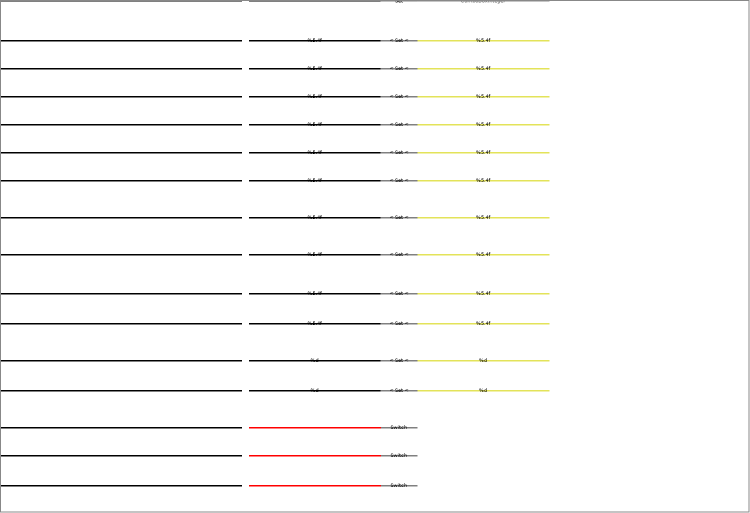
VISUALIZATION Visu_Mparam_Cool  // 750x513
    Frame (0,40 750x28)
        shows Param_LREAL(nIdx := 4)
    Frame (0,68 750x28)
        shows Param_LREAL(nIdx := 6)
    Frame (0,96 750x28)
        shows Param_LREAL(nIdx := 8)
    Frame (0,124 750x28)
        shows Param_LREAL(nIdx := 10)
    Frame (0,360 750x28)
        shows Param_DINT(nIdx := 11)
    Frame (0,0 750x28)
        shows Param_ENUM_SelOut(nIdx := GlobalOne)
    Frame (0,152 750x28)
        shows Param_LREAL(nIdx := 16)
    Frame (0,180 750x28)
        shows Param_LREAL(nIdx := 17)
    Frame (0,217 750x28)
        shows Param_LREAL(nIdx := 21)
    Frame (0,293 750x28)
        shows Param_LREAL(nIdx := 37)
    Frame (0,323 750x28)
        shows Param_LREAL(nIdx := 38)
    Frame (0,427 750x28)
        shows Param_BOOL(nIdx := GlobalOne)
    Frame (0,455 750x28)
        shows Param_BOOL(nIdx := 3)
    Frame (0,485 750x28)
        shows Param_BOOL(nIdx := 18)
    Frame (0,254 750x28)
        shows Param_LREAL(nIdx := 32)
    Frame (0,390 750x28)
        shows Param_DINT(nIdx := 12)
END_VISUALIZATION

// ---- Temperature/VISUs/VISUs/Pages/Machine/Subpage/Visu_Mparam_Extruder.TcVIS
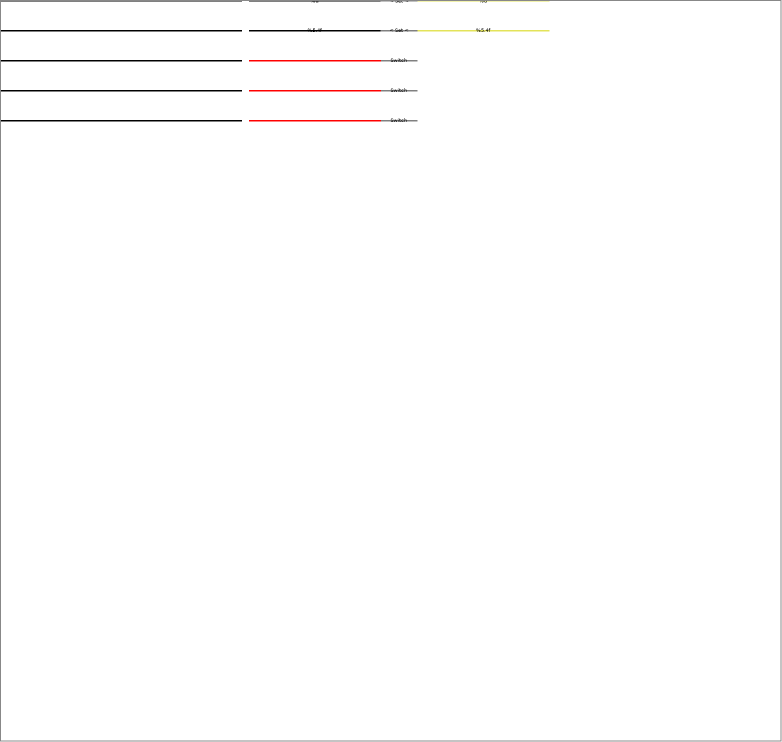
VISUALIZATION Visu_Mparam_Extruder  // 782x742
    Frame (0,30 750x30)
        shows Param_LREAL(nIdx := 3)
    Frame (0,90 750x30)
        shows Param_BOOL(nIdx := 8)
    Frame (0,60 750x30)
        shows Param_BOOL(nIdx := 2)
    Frame (0,0 750x30)
        shows Param_DINT(nIdx := 3)
    Frame (0,120 750x30)
        shows Param_BOOL(nIdx := 14)
    Rectangle (30,710 750x30)
END_VISUALIZATION

// ---- Temperature/VISUs/VISUs/Pages/Machine/Subpage/Visu_Mparam_General.TcVIS
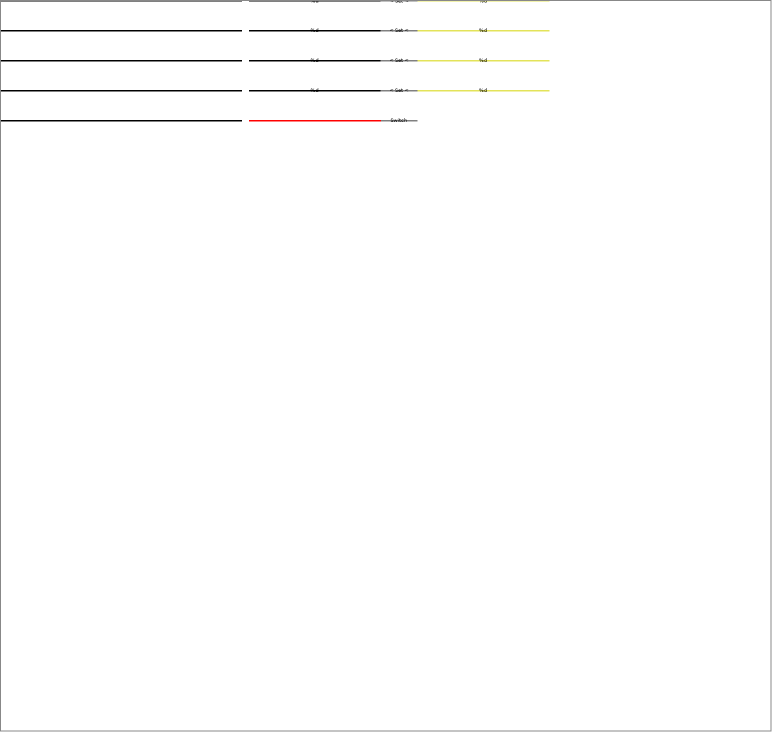
VISUALIZATION Visu_Mparam_General  // 772x732
    Frame (0,120 750x30)
        shows Param_BOOL(nIdx := 6)
    Frame (0,0 750x30)
        shows Param_DINT(nIdx := 3)
    Frame (0,30 750x30)
        shows Param_DINT(nIdx := 4)
    Frame (0,60 750x30)
        shows Param_DINT(nIdx := 5)
    Frame (0,90 750x30)
        shows Param_DINT(nIdx := 6)
    Rectangle (10,690 750x30)
    Rectangle (20,700 750x30)
END_VISUALIZATION

// ---- Temperature/VISUs/VISUs/Pages/Machine/Subpage/Visu_Mparam_Heat.TcVIS
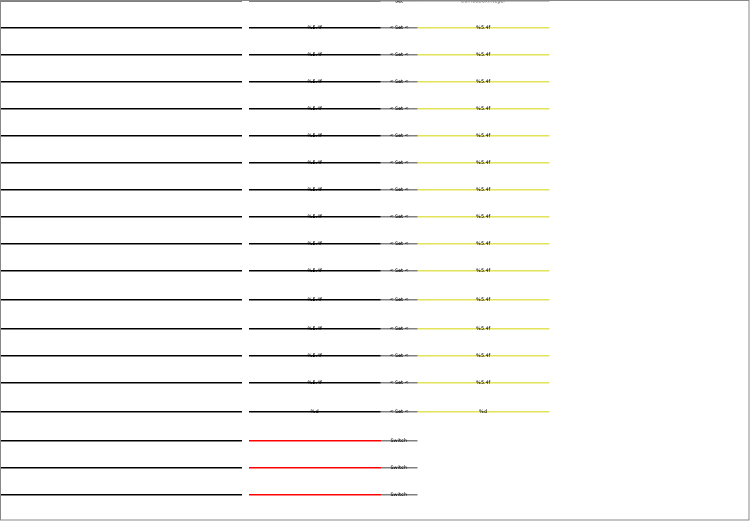
VISUALIZATION Visu_Mparam_Heat  // 750x521
    Frame (0,27 750x27)
        shows Param_LREAL(nIdx := 5)
    Frame (0,54 750x27)
        shows Param_LREAL(nIdx := 7)
    Frame (0,81 750x27)
        shows Param_LREAL(nIdx := 9)
    Frame (0,108 750x27)
        shows Param_LREAL(nIdx := 11)
    Frame (0,411 750x27)
        shows Param_DINT(nIdx := 10)
    Frame (0,0 750x27)
        shows Param_ENUM_SelOut(nIdx := 2)
    Frame (0,135 750x27)
        shows Param_LREAL(nIdx := 12)
    Frame (0,162 750x27)
        shows Param_LREAL(nIdx := 13)
    Frame (0,189 750x27)
        shows Param_LREAL(nIdx := 14)
    Frame (0,216 750x27)
        shows Param_LREAL(nIdx := 15)
    Frame (0,243 750x27)
        shows Param_LREAL(nIdx := 17)
    Frame (0,270 750x27)
        shows Param_LREAL(nIdx := 18)
    Frame (0,299 750x27)
        shows Param_LREAL(nIdx := 22)
    Frame (0,328 750x27)
        shows Param_LREAL(nIdx := 33)
    Frame (0,355 750x27)
        shows Param_LREAL(nIdx := 34)
    Frame (0,382 750x27)
        shows Param_LREAL(nIdx := 36)
    Frame (0,440 750x27)
        shows Param_BOOL(nIdx := 12)
    Frame (0,467 750x27)
        shows Param_BOOL(nIdx := 16)
    Frame (0,494 750x27)
        shows Param_BOOL(nIdx := 19)
END_VISUALIZATION

// ---- Temperature/VISUs/VISUs/Pages/Machine/Subpage/Visu_Mparam_Supply.TcVIS
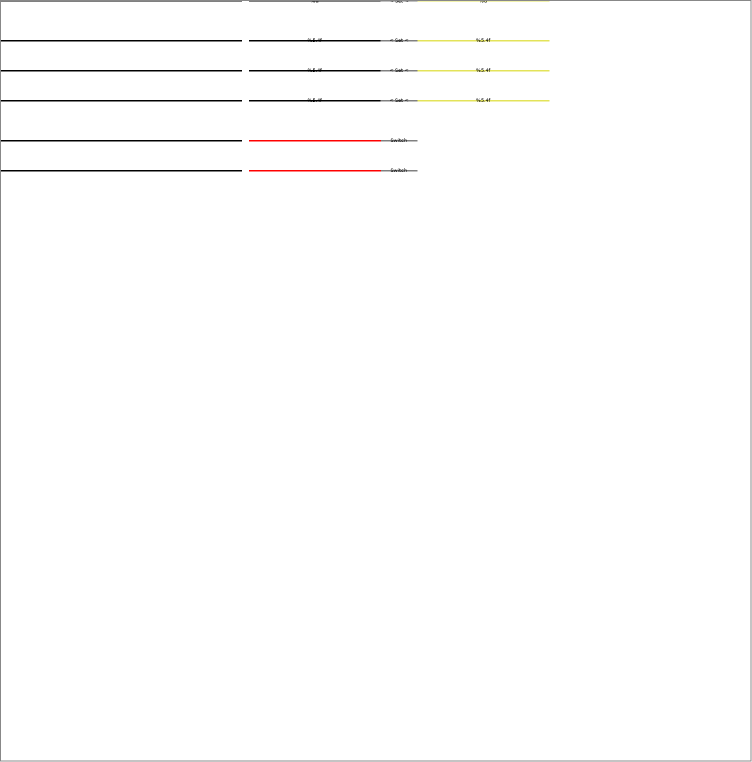
VISUALIZATION Visu_Mparam_Supply  // 752x762
    Frame (0,40 750x30)
        shows Param_LREAL(nIdx := 21)
    Frame (0,70 750x30)
        shows Param_LREAL(nIdx := 22)
    Frame (0,100 750x30)
        shows Param_LREAL(nIdx := 23)
    Frame (0,0 750x30)
        shows Param_DINT(nIdx := 6)
    Frame (0,140 750x30)
        shows Param_BOOL(nIdx := 11)
    Frame (0,170 750x30)
        shows Param_BOOL(nIdx := 15)
    Rectangle (0,730 750x30)
END_VISUALIZATION

// ---- Temperature/VISUs/VISUs/Pages/Machine/Subpage/Visu_Mparam_Temperature.TcVIS
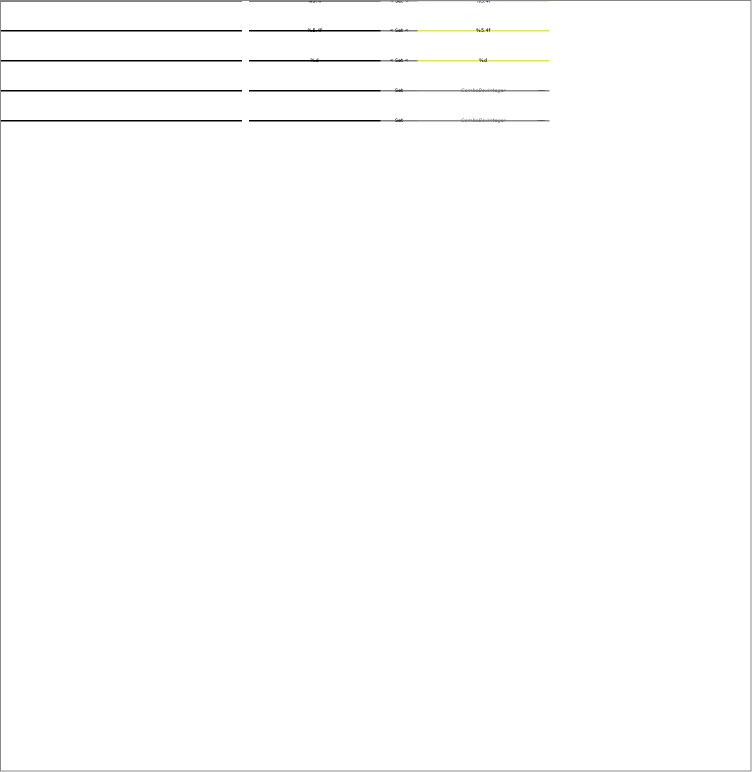
VISUALIZATION Visu_Mparam_Temperature  // 752x772
    Frame (0,0 750x30)
        shows Param_LREAL(nIdx := GlobalOne)
    Frame (0,30 750x30)
        shows Param_LREAL(nIdx := 2)
    Frame (0,60 750x30)
        shows Param_DINT(nIdx := 9)
    Frame (0,90 750x30)
        shows Param_ENUM_TermType(nIdx := 3)
    Frame (0,120 750x30)
        shows Param_ENUM_SensType(nIdx := 4)
    Rectangle (0,740 750x30)
END_VISUALIZATION

// ---- Temperature/VISUs/VISUs/Pages/Machine/Visu_MParam.TcVIS
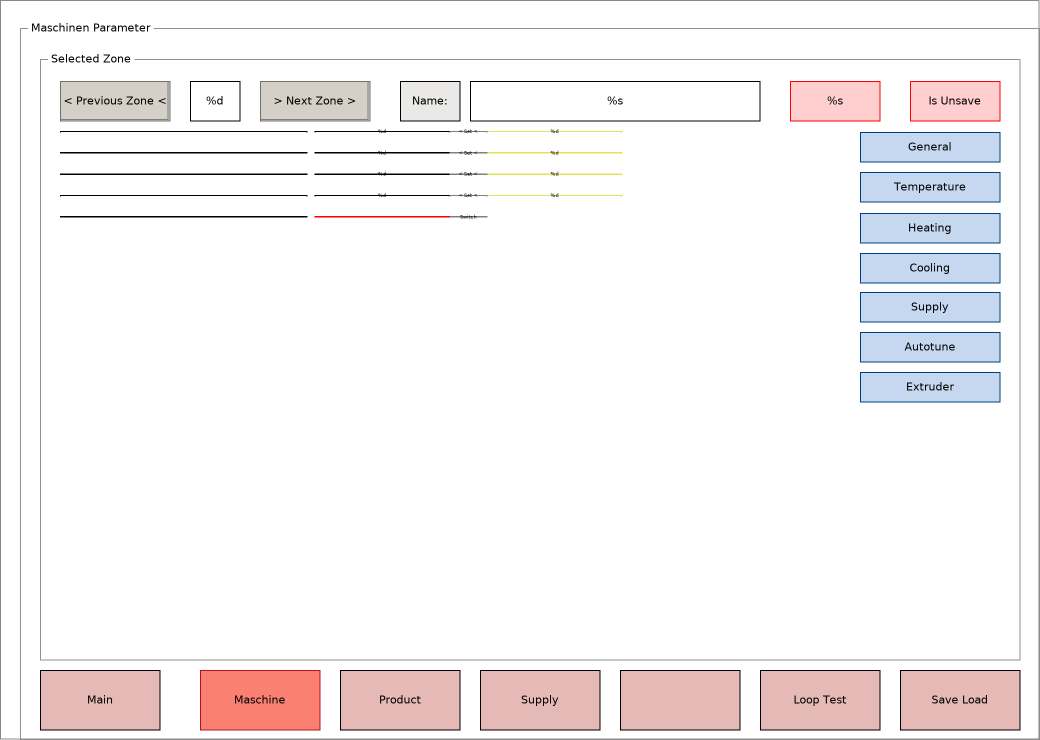
VISUALIZATION Visu_MParam  // 1040x740
    GroupBox (20,20 1020x720), "Maschinen Parameter"
        Rectangle (20,650 120x60), "Main"
            OnMouseClick: change screen: Visu_Main
        Rectangle (880,650 120x60), "Save Load"
            OnMouseClick: change screen: Visu_SaveLoad
        Rectangle (320,650 120x60), "Product"
            OnMouseClick: change screen: Visu_PParam
        Rectangle (180,650 120x60), "Maschine"
            OnMouseClick: change screen: Visu_MParam
        Rectangle (460,650 120x60), "Supply"
            OnMouseClick: change screen: Visu_Supply
        Rectangle (600,650 120x60)
        GroupBox (20,31 980x609), "Selected Zone"
            Rectangle (150,30 50x40), "%d", text variable: nVisuCount
            Button (20,30 110x40), "< Previous Zone <"
                tap bVisuBefore
            Button (220,30 110x40), "> Next Zone >"
                tap bVisuNext
            Rectangle (750,30 90x40), "%s", text variable: stMParam_Visu.sInUse, colour toggle: aaaPfwTempMparamFromHmi[nVisuCount].InUse
                OnMouseClick: toggle aaaPfwTempMparamFromHmi[nVisuCount].InUse
                OnMouseClick: execute { stParamsUnsave.mParams[nVisuCount]:=TRUE; }
            Rectangle (430,30 290x40), "%s", text variable: aaaPfwTempMparamFromHmi[nVisuCount].ZoneName
                OnMouseClick: write the text variable via Edit
                OnMouseClick: execute { stParamsUnsave.mParams[nVisuCount]:=TRUE; }
            Rectangle (360,30 60x40), "Name:"
            Rectangle (870,30 90x40), "Is Unsave", invisible if: Not stParamsUnsave.mParams[nVisuCount]
                OnMouseClick: execute { aaaPfwTempMparamFromHmi[nVisuCount].SaveDelay:=1000; stParamsUnsave.mParams[nVisuCount]:=FALSE; }
            Rectangle (820,81 140x30), "General", colour toggle: stMParam_Visu.nActiveParamList=0
                OnMouseClick: execute { stMParam_Visu.nActiveParamList:=0; }
            Frame (20,80 790x521), frame switch variable: stMParam_Visu.nActiveParamList
                shows Visu_Mparam_General()
                shows Visu_Mparam_Temperature()
                shows Visu_Mparam_Heat()
                shows Visu_Mparam_Cool()
                shows Visu_Mparam_Supply()
                shows Visu_Mparam_Autotune()
                shows Visu_Mparam_Extruder()
            Rectangle (820,202 140x30), "Cooling", colour toggle: stMParam_Visu.nActiveParamList=3
                OnMouseClick: execute { stMParam_Visu.nActiveParamList:=3; }
            Rectangle (820,162 140x30), "Heating", colour toggle: stMParam_Visu.nActiveParamList=2
                OnMouseClick: execute { stMParam_Visu.nActiveParamList:=2; }
            Rectangle (820,321 140x30), "Extruder", colour toggle: stMParam_Visu.nActiveParamList=6, invisible if: NOT MAIN.bFirstCycle
                OnMouseClick: execute { stMParam_Visu.nActiveParamList:=6; }
            Rectangle (820,281 140x30), "Autotune", colour toggle: stMParam_Visu.nActiveParamList=5
                OnMouseClick: execute { stMParam_Visu.nActiveParamList:=5; }
            Rectangle (820,241 140x30), "Supply", colour toggle: stMParam_Visu.nActiveParamList=4
                OnMouseClick: execute { stMParam_Visu.nActiveParamList:=4; }
            Rectangle (820,121 140x30), "Temperature", colour toggle: stMParam_Visu.nActiveParamList=1
                OnMouseClick: execute { stMParam_Visu.nActiveParamList:=1; }
        Rectangle (740,650 120x60), "Loop Test"
            OnMouseClick: change screen: Visu_LoopTest
END_VISUALIZATION

// ---- Temperature/VISUs/VISUs/Pages/Product/Param_LREAL_Pparam.TcVIS
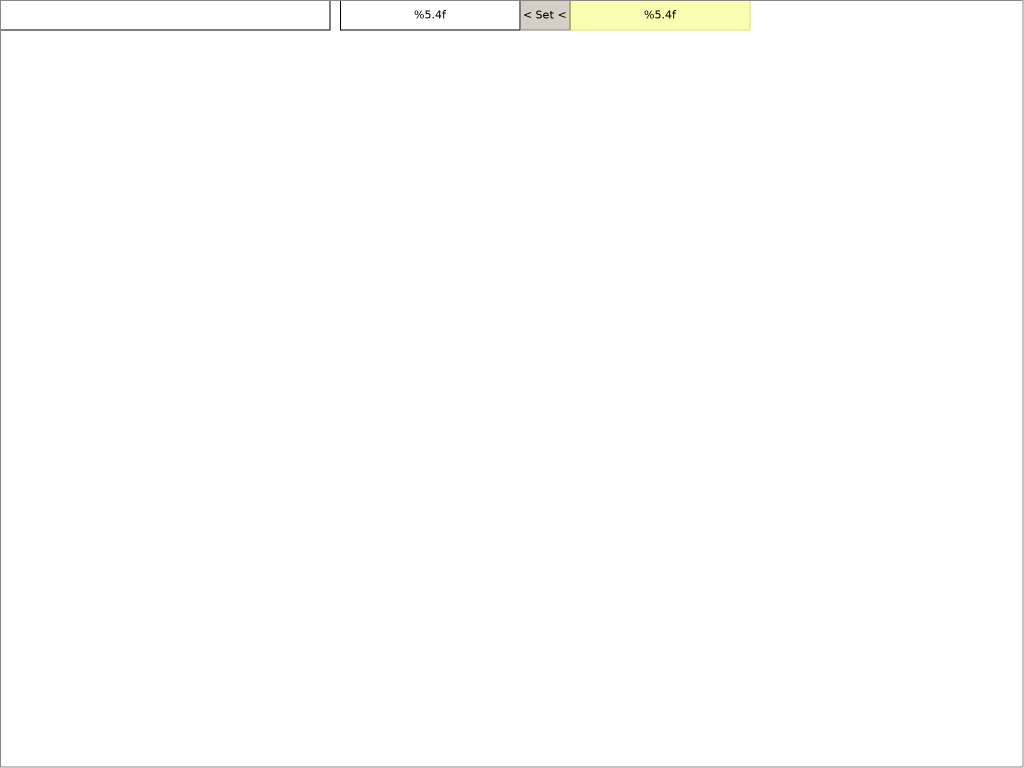
VISUALIZATION Param_LREAL_Pparam  // 1024x768
    Rectangle (340,0 180x30), "%5.4f", text variable: stPParam_Visu.fLrealAktValue[nIdx]
    Rectangle (0,0 330x30), text list: 'TL_Pparmas', text index: nIdx
    Rectangle (570,0 180x30), "%5.4f", text variable: stPParam_Visu.fLrealNewValue[nIdx]
        OnMouseClick: write the text variable via Default
    Rectangle (520,0 50x30), "< Set <"
        OnMouseClick: execute { stPParam_Visu.bLrealSetValue[nIdx]:=TRUE; }
END_VISUALIZATION

// ---- Temperature/VISUs/VISUs/Pages/Product/Visu_PParam.TcVIS
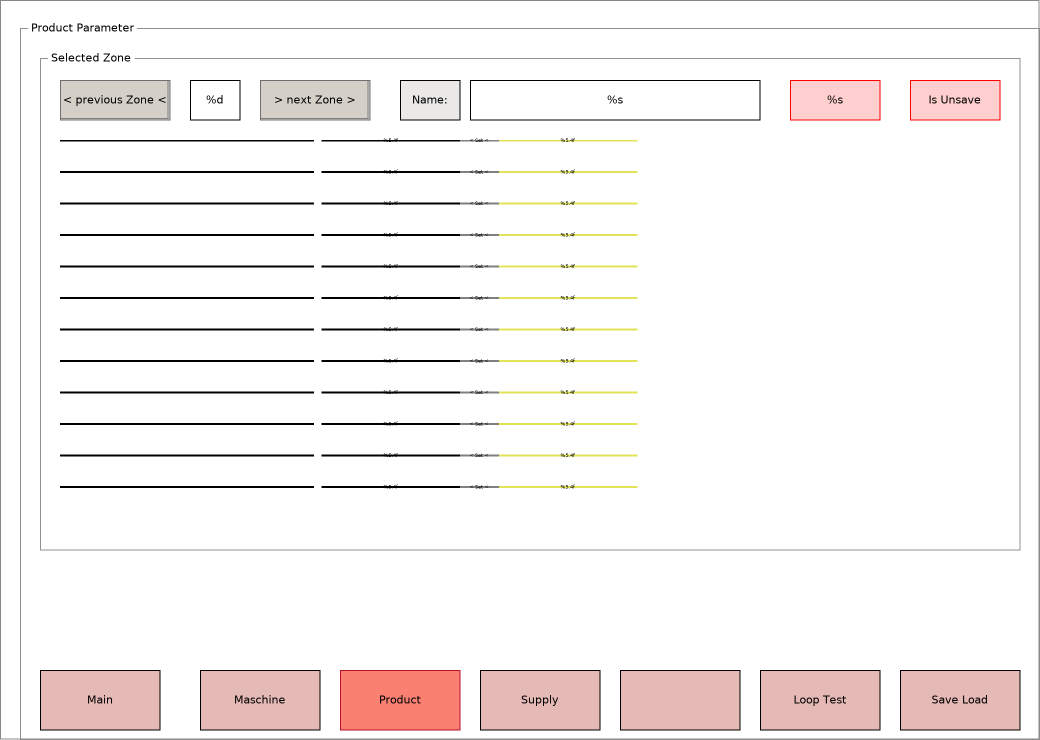
VISUALIZATION Visu_PParam  // 1040x740
    GroupBox (20,20 1020x720), "Product Parameter"
        Rectangle (20,650 120x60), "Main"
            OnMouseClick: change screen: Visu_Main
        Rectangle (880,650 120x60), "Save Load"
            OnMouseClick: change screen: Visu_SaveLoad
        Rectangle (320,650 120x60), "Product"
            OnMouseClick: change screen: Visu_PParam
        GroupBox (20,30 980x500), "Selected Zone"
            Rectangle (150,30 50x40), "%d", text variable: nVisuCount
            Button (20,30 110x40), "< previous Zone <"
                tap bVisuBefore
            Button (220,30 110x40), "> next Zone >"
                tap bVisuNext
            Rectangle (430,30 290x40), "%s", text variable: aaaPfwTempMparamFromHmi[nVisuCount].ZoneName
            Rectangle (360,30 60x40), "Name:"
            Frame (20,90 790x380)
                shows Visu_PParam_Params()
                shows Visu_MParam_ENUM()
                shows Visu_MParam_BOOL()
                shows Visu_MParam_INT()
            Rectangle (870,30 90x40), "Is Unsave", invisible if: Not stParamsUnsave.pParams[nVisuCount]
                OnMouseClick: execute { aaaPfwTempPparamFromHmi[nVisuCount].SaveDelay:=1000; stParamsUnsave.pParams[nVisuCount]:=FALSE; }
        Rectangle (180,650 120x60), "Maschine"
            OnMouseClick: change screen: Visu_MParam
    Rectangle (480,670 120x60), "Supply"
        OnMouseClick: change screen: Visu_Supply
    Rectangle (620,670 120x60)
    Rectangle (760,670 120x60), "Loop Test"
        OnMouseClick: change screen: Visu_LoopTest
    Rectangle (790,80 90x40), "%s", text variable: stMParam_Visu.sInUse, colour toggle: aaaPfwTempMparamFromHmi[nVisuCount].InUse
        OnMouseClick: toggle aaaPfwTempMparamFromHmi[nVisuCount].InUse
        OnMouseClick: execute { stParamsUnsave.mParams[nVisuCount]:=TRUE; }
END_VISUALIZATION

// ---- Temperature/VISUs/VISUs/Pages/Product/Visu_PParam_Params.TcVIS
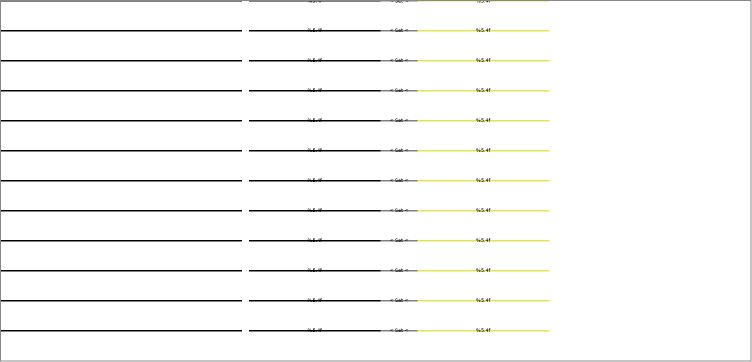
VISUALIZATION Visu_PParam_Params  // 752x362
    Frame (0,0 750x30)
        shows Param_LREAL_Pparam(nIdx := GlobalOne)
    Frame (0,30 750x30)
        shows Param_LREAL_Pparam(nIdx := 2)
    Frame (0,60 750x30)
        shows Param_LREAL_Pparam(nIdx := 3)
    Frame (0,90 750x30)
        shows Param_LREAL_Pparam(nIdx := 4)
    Frame (0,120 750x30)
        shows Param_LREAL_Pparam(nIdx := 5)
    Frame (0,150 750x30)
        shows Param_LREAL_Pparam(nIdx := 6)
    Frame (0,180 750x30)
        shows Param_LREAL_Pparam(nIdx := 7)
    Frame (0,210 750x30)
        shows Param_LREAL_Pparam(nIdx := 8)
    Frame (0,240 750x30)
        shows Param_LREAL_Pparam(nIdx := 9)
    Frame (0,270 750x30)
        shows Param_LREAL_Pparam(nIdx := 10)
    Frame (0,300 750x30)
        shows Param_LREAL_Pparam(nIdx := 11)
    Frame (0,330 750x30)
        shows Param_LREAL_Pparam(nIdx := 12)
END_VISUALIZATION

// ---- Temperature/VISUs/VISUs/Pages/Supply/Param_LREAL_Supply.TcVIS
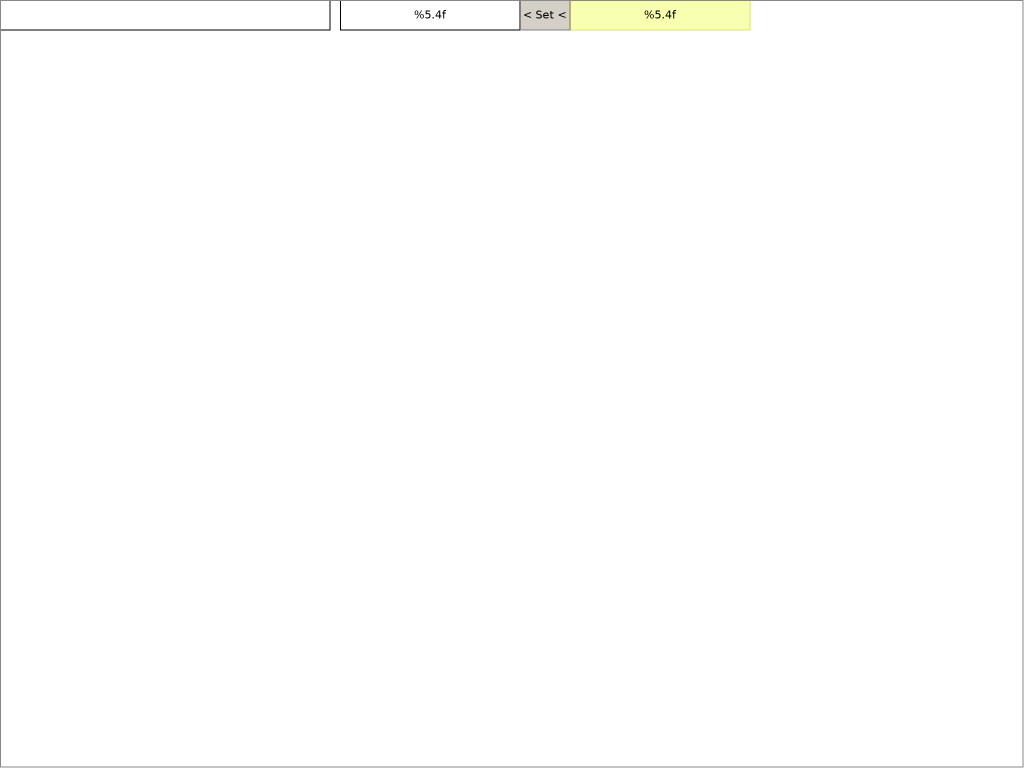
VISUALIZATION Param_LREAL_Supply  // 1024x768
    Rectangle (340,0 180x30), "%5.4f", text variable: stSupply_Visu.fLrealAktValue[nIdx]
    Rectangle (0,0 330x30), text list: 'TL_Supply', text index: nIdx
    Rectangle (570,0 180x30), "%5.4f", text variable: stSupply_Visu.fLrealNewValue[nIdx]
        OnMouseClick: write the text variable via Default
    Rectangle (520,0 50x30), "< Set <"
        OnMouseClick: execute { stSupply_Visu.bLrealSetValue[nIdx]:=TRUE; }
END_VISUALIZATION

// ---- Temperature/VISUs/VISUs/Pages/Supply/Visu_Supply.TcVIS
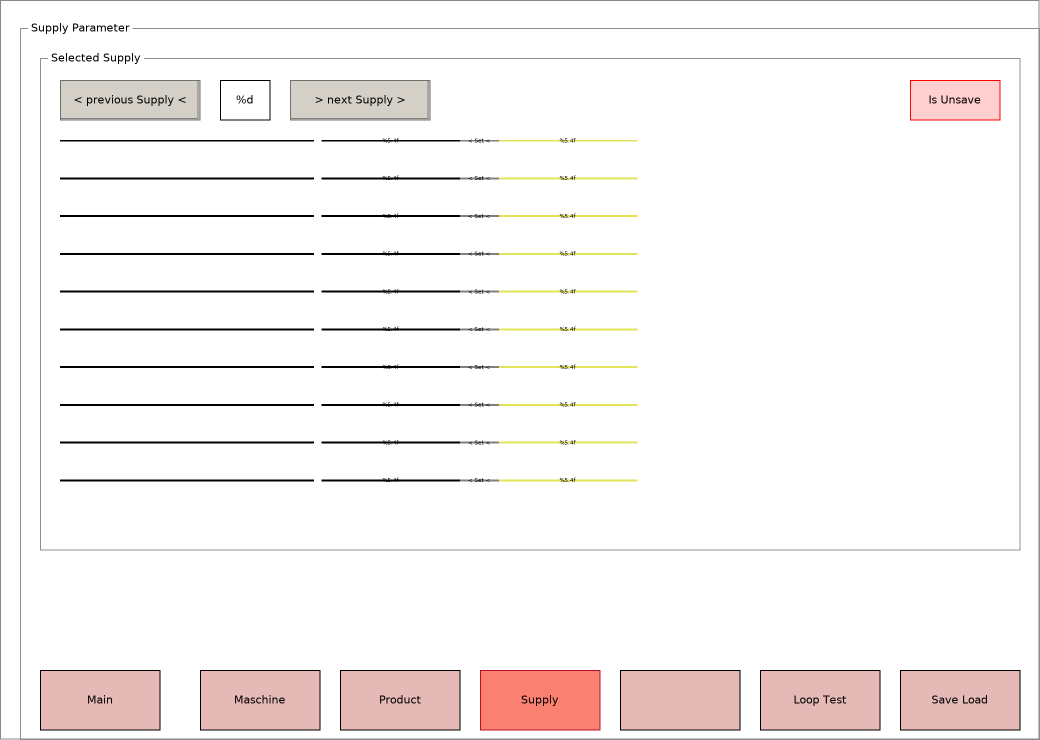
VISUALIZATION Visu_Supply  // 1040x740
    GroupBox (20,20 1020x720), "Supply Parameter"
        Rectangle (20,650 120x60), "Main"
            OnMouseClick: change screen: Visu_Main
        Rectangle (880,650 120x60), "Save Load"
            OnMouseClick: change screen: Visu_SaveLoad
        Rectangle (320,650 120x60), "Product"
            OnMouseClick: change screen: Visu_PParam
        Rectangle (180,650 120x60), "Maschine"
            OnMouseClick: change screen: Visu_MParam
        Rectangle (460,650 120x60), "Supply"
            OnMouseClick: change screen: Visu_Supply
        Rectangle (600,650 120x60)
        Rectangle (740,650 120x60), "Loop Test"
            OnMouseClick: change screen: Visu_LoopTest
        GroupBox (20,30 980x500), "Selected Supply"
            Rectangle (180,30 50x40), "%d", text variable: nSupplyCnt
            Button (20,30 140x40), "< previous Supply <"
                OnMouseClick: execute { nSupplyCnt:= MAX(cnPfwAppSupplyFirst, nSupplyCnt-1); }
            Button (250,30 140x40), "> next Supply >"
                OnMouseClick: execute { nSupplyCnt:= MIN(cnPfwAppSupplyLast, nSupplyCnt+1); }
            Rectangle (870,30 90x40), "Is Unsave", invisible if: Not stParamsUnsave.supply[nSupplyCnt]
                OnMouseClick: execute { stPfwSupplyLineCfg[nSupplyCnt].SaveDelay:=1000; stParamsUnsave.supply[nSupplyCnt]:=FALSE; }
            Frame (20,90 790x380)
                shows Visu_Supply_Params()
                shows Visu_MParam_ENUM()
                shows Visu_MParam_BOOL()
                shows Visu_MParam_INT()
END_VISUALIZATION

// ---- Temperature/VISUs/VISUs/Pages/Supply/Visu_Supply_Params.TcVIS
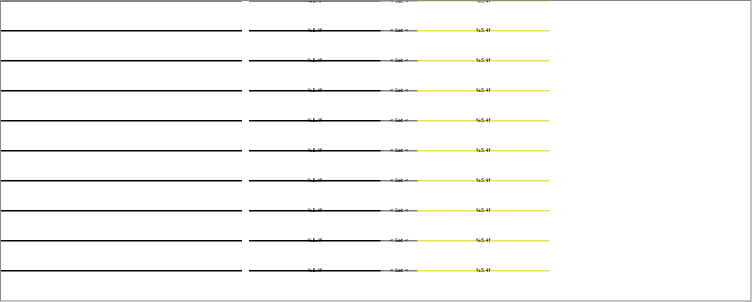
VISUALIZATION Visu_Supply_Params  // 752x302
    Frame (0,0 750x30)
        shows Param_LREAL_Supply(nIdx := GlobalOne)
    Frame (0,30 750x30)
        shows Param_LREAL_Supply(nIdx := 2)
    Frame (0,60 750x30)
        shows Param_LREAL_Supply(nIdx := 3)
    Frame (0,120 750x30)
        shows Param_LREAL_Supply(nIdx := 5)
    Frame (0,90 750x30)
        shows Param_LREAL_Supply(nIdx := 4)
    Frame (0,270 750x30)
        shows Param_LREAL_Supply(nIdx := 10)
    Frame (0,240 750x30)
        shows Param_LREAL_Supply(nIdx := 9)
    Frame (0,210 750x30)
        shows Param_LREAL_Supply(nIdx := 8)
    Frame (0,180 750x30)
        shows Param_LREAL_Supply(nIdx := 7)
    Frame (0,150 750x30)
        shows Param_LREAL_Supply(nIdx := 6)
END_VISUALIZATION

// ---- Temperature/VISUs/VISUs/Pages/Visu_Main.TcVIS
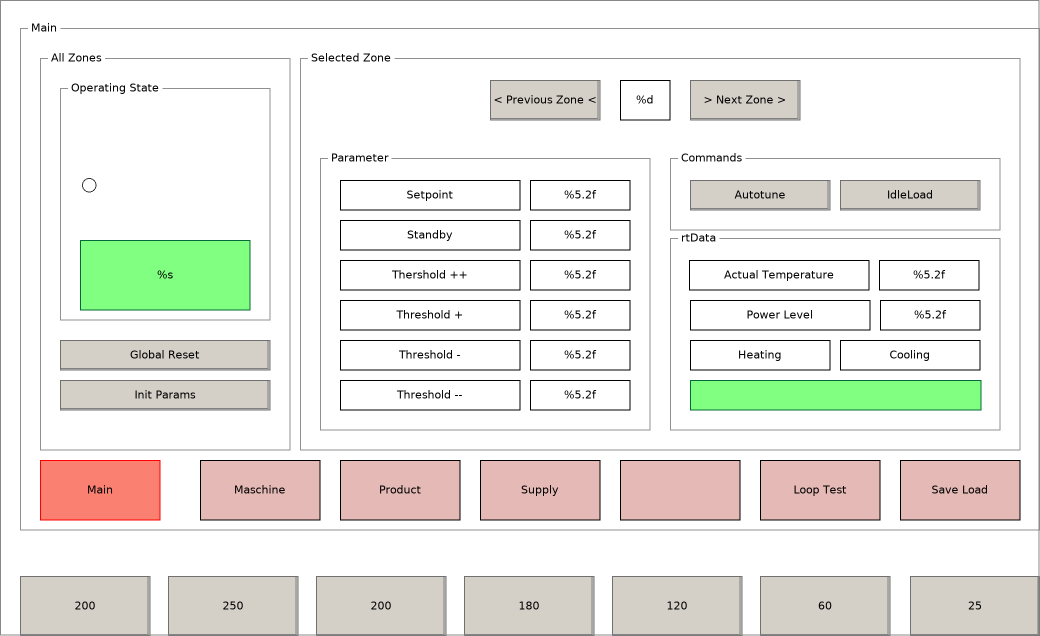
VISUALIZATION Visu_Main  // 1040x636
    GroupBox (20,20 1020x510), "Main"
        Rectangle (20,440 120x60), "Main"
            OnMouseClick: change screen: Visu_Main
        Rectangle (880,440 120x60), "Save Load"
            OnMouseClick: change screen: Visu_SaveLoad
        Rectangle (320,440 120x60), "Product"
            OnMouseClick: change screen: Visu_PParam
        Rectangle (180,440 120x60), "Maschine"
            OnMouseClick: change screen: Visu_MParam
    GroupBox (40,50 250x400), "All Zones", input disabled if: TemperatureCtrl.eState<>eMainSM_Idle
        GroupBox (20,30 210x240), "Operating State", input disabled if: TemperatureCtrl.eState<>eMainSM_Idle
            RadioButton (20,30 150x150), variable: eStatus
                Areas[0]: Text=Off
                Areas[1]: Text=Standby
                Areas[2]: Text=On
                Areas[3]: Text=Autotune
                Areas[4]: Text=Idle Load
            Rectangle (20,160 170x70), "%s", text variable: sErrorText, colour toggle: bGlobalError
        Button (20,330 210x30), "Init Params"
            tap bParamsInit
        Button (20,290 210x30), "Global Reset"
            tap aaaTempFault_Reset
    GroupBox (300,50 720x400), "Selected Zone"
        Rectangle (320,30 50x40), "%d", text variable: nVisuCount
        Button (190,30 110x40), "< Previous Zone <"
            tap bVisuBefore
        Button (390,30 110x40), "> Next Zone >"
            tap bVisuNext
        GroupBox (20,100 330x280), "Parameter"
            Rectangle (20,30 180x30), "Setpoint"
            Rectangle (20,70 180x30), "Standby"
            Rectangle (20,110 180x30), "Thershold ++"
            Rectangle (20,150 180x30), "Threshold +"
            Rectangle (20,190 180x30), "Threshold -"
            Rectangle (20,230 180x30), "Threshold --"
            Rectangle (210,30 100x30), "%5.2f", text variable: aaaPfwTempPparamFromHmi[nVisuCount].Setpoint
            Rectangle (210,70 100x30), "%5.2f", text variable: aaaPfwTempPparamFromHmi[nVisuCount].StandbySetpoint
            Rectangle (210,110 100x30), "%5.2f", text variable: aaaPfwTempPparamFromHmi[nVisuCount].Threshold_PP
            Rectangle (210,150 100x30), "%5.2f", text variable: aaaPfwTempPparamFromHmi[nVisuCount].Threshold_P
            Rectangle (210,190 100x30), "%5.2f", text variable: aaaPfwTempPparamFromHmi[nVisuCount].Threshold_M
            Rectangle (210,230 100x30), "%5.2f", text variable: aaaPfwTempPparamFromHmi[nVisuCount].Threshold_MM
        GroupBox (370,180 330x200), "rtData"
            Rectangle (210,70 100x30), "%5.2f", text variable: aaaPfwTempToHmi[nVisuCount].PowerLevel
            Rectangle (19,30 180x30), "Actual Temperature"
            Rectangle (209,30 100x30), "%5.2f", text variable: aaaPfwTempToHmi[nVisuCount].ActualTemp
            Rectangle (20,70 180x30), "Power Level"
            Rectangle (170,110 140x30), "Cooling", colour toggle: aaaPfwTempToHmi[nVisuCount].Cooling
            Rectangle (20,110 140x30), "Heating", colour toggle: aaaPfwTempToHmi[nVisuCount].Heating
            Rectangle (20,150 291x30), colour toggle: aaaPfwTempToHmi[nVisuCount].Error, text list: 'TL_TcPfw_ErrorId', text index: INT_TO_STRING(aaaPfwTempToHmi[nVisuCount].ErrorId)
                OnMouseClick: ChangeLanguage ChangeLanguage=en
        GroupBox (370,100 330x80), "Commands", input disabled if: aaaPfwTempMparamFromHmi[nVisuCount].Autotune OR aaaPfwTempMparamFromHmi[nVisuCount].Ena_TuneIdleLoad OR TemperatureCtrl.eState<>eMainSM_Idle
            Button (20,30 140x30), "Autotune"
                tap bVisuAutotune
            Button (170,30 140x30), "IdleLoad"
                tap bVisuIdleLoad
    Rectangle (480,460 120x60), "Supply"
        OnMouseClick: change screen: Visu_Supply
    Rectangle (620,460 120x60)
    Rectangle (760,460 120x60), "Loop Test"
        OnMouseClick: change screen: Visu_LoopTest
    Button (20,576 130x60), "200"
        OnMouseUp: execute { aaaPfwTempPparamFromHmi[1].Setpoint:= 200; }
    Button (168,576 130x60), "250"
        OnMouseUp: execute { aaaPfwTempPparamFromHmi[1].Setpoint:= 250; }
    Button (316,576 130x60), "200"
        OnMouseUp: execute { aaaPfwTempPparamFromHmi[1].Setpoint:= 200; }
    Button (464,576 130x60), "180"
        OnMouseUp: execute { aaaPfwTempPparamFromHmi[1].Setpoint:= 180; }
    Button (612,576 130x60), "120"
        OnMouseUp: execute { aaaPfwTempPparamFromHmi[1].Setpoint:= 120; }
    Button (760,576 130x60), "60"
        OnMouseUp: execute { aaaPfwTempPparamFromHmi[1].Setpoint:= 60; }
    Button (910,576 130x60), "25"
        OnMouseUp: execute { aaaPfwTempPparamFromHmi[1].Setpoint:= 25; }
END_VISUALIZATION
